LIN {X 0,Y 358.147,Z 231.366,A -85,B 0,C 180,E1 16534.491,E2 16534.491} C_VEL
LIN {X 0,Y 360.808,Z 235.237,A -85,B 0,C 180,E1 16533.457,E2 16533.457} C_VEL
LIN {X 0,Y 363.287,Z 237.581,A -85,B 0,C 180,E1 16532.591,E2 16532.591} C_VEL
LIN {X 0,Y 366.593,Z 241.883,A -85,B 0,C 180,E1 16531.445,E2 16531.445} C_VEL
LIN {X 0,Y 368.213,Z 243.704,A -85,B 0,C 180,E1 16530.917,E2 16530.917} C_VEL
LIN {X 0,Y 371.953,Z 248.281,A -85,B 0,C 180,E1 16529.732,E2 16529.732} C_VEL
LIN {X 0,Y 377.988,Z 256.41,A -85,B 0,C 180,E1 16527.924,E2 16527.924} C_VEL
LIN {X 0,Y 386.57,Z 269.394,A -85,B 0,C 180,E1 16525.541,E2 16525.541} C_VEL
LIN {X 0,Y 395.488,Z 283.924,A -85,B 0,C 180,E1 16523.278,E2 16523.278} C_VEL
LIN {X 0,Y 404.338,Z 299.581,A -85,B 0,C 180,E1 16521.202,E2 16521.202} C_VEL
LIN {X 0,Y 413.977,Z 318.387,A -85,B 0,C 180,E1 16519.091,E2 16519.091} C_VEL
LIN {X 0,Y 416.532,Z 324.265,A -85,B 0,C 180,E1 16518.54,E2 16518.54} C_VEL
LIN {X 0,Y 406.024,Z 519.661,A -85,B 0,C 180,E1 16515.165,E2 16515.165} C_VEL
LIN {X 0,Y 404.264,Z 537.979,A -85,B 0,C 180,E1 16514.727,E2 16514.727} C_VEL
LIN {X 0,Y 401.335,Z 559.6,A -85,B 0,C 180,E1 16514.028,E2 16514.028} C_VEL
LIN {X 0,Y 397.456,Z 581.194,A -85,B 0,C 180,E1 16513.057,E2 16513.057} C_VEL
LIN {X 0,Y 393.804,Z 598.492,A -85,B 0,C 180,E1 16512.084,E2 16512.084} C_VEL
LIN {X 0,Y 389.995,Z 614.356,A -85,B 0,C 180,E1 16511.015,E2 16511.015} C_VEL
LIN {X 0,Y 385.902,Z 629.8,A -85,B 0,C 180,E1 16509.784,E2 16509.784} C_VEL
LIN {X 0,Y 381.564,Z 644.781,A -85,B 0,C 180,E1 16508.387,E2 16508.387} C_VEL
LIN {X 0,Y 376.69,Z 660.514,A -85,B 0,C 180,E1 16506.667,E2 16506.667} C_VEL
LIN {X 0,Y 370.561,Z 678.911,A -85,B 0,C 180,E1 16504.243,E2 16504.243} C_VEL
LIN {X 0,Y 365.986,Z 691.98,A -85,B 0,C 180,E1 16502.186,E2 16502.186} C_VEL
LIN {X 0,Y 361.741,Z 703.869,A -85,B 0,C 180,E1 16500.015,E2 16500.015} C_VEL
LIN {X 0,Y 357.987,Z 714.365,A -85,B 0,C 180,E1 16497.8,E2 16497.8} C_VEL
LIN {X 0,Y 354.508,Z 724.257,A -85,B 0,C 180,E1 16495.382,E2 16495.382} C_VEL
LIN {X 0,Y 351.404,Z 733.441,A -85,B 0,C 180,E1 16492.763,E2 16492.763} C_VEL
LIN {X 0,Y 348.508,Z 742.76,A -85,B 0,C 180,E1 16489.611,E2 16489.611} C_VEL
LIN {X 0,Y 346.148,Z 751.408,A -85,B 0,C 180,E1 16485.925,E2 16485.925} C_VEL
LIN {X 0,Y 344.933,Z 757.022,A -85,B 0,C 180,E1 16482.896,E2 16482.896} C_VEL
LIN {X 0,Y 344.287,Z 761.191,A -85,B 0,C 180,E1 16480.034,E2 16480.034} C_VEL
LIN {X 0,Y 343.998,Z 764.291,A -85,B 0,C 180,E1 16477.179,E2 16477.179} C_VEL
LIN {X 0,Y 343.938,Z 766.265,A -85,B 0,C 180,E1 16474.501,E2 16474.501} C_VEL
LIN {X 0,Y 343.961,Z 767.366,A -85,B 0,C 180,E1 16471.666,E2 16471.666} C_VEL
LIN {X 0,Y 343.968,Z 767.484,A -85,B 0,C 180,E1 16469.001,E2 16469.001} C_VEL
LIN {X 0,Y 343.943,Z 766.62,A -85,B 0,C 180,E1 16466.167,E2 16466.167} C_VEL
LIN {X 0,Y 343.979,Z 764.736,A -85,B 0,C 180,E1 16463.324,E2 16463.324} C_VEL
LIN {X 0,Y 344.211,Z 761.817,A -85,B 0,C 180,E1 16460.47,E2 16460.47} C_VEL
LIN {X 0,Y 344.79,Z 757.833,A -85,B 0,C 180,E1 16457.61,E2 16457.61} C_VEL
LIN {X 0,Y 345.827,Z 752.744,A -85,B 0,C 180,E1 16454.748,E2 16454.748} C_VEL
LIN {X 0,Y 347.309,Z 746.894,A -85,B 0,C 180,E1 16452.061,E2 16452.061} C_VEL
LIN {X 0,Y 349.33,Z 739.94,A -85,B 0,C 180,E1 16449.387,E2 16449.387} C_VEL
LIN {X 0,Y 351.939,Z 731.816,A -85,B 0,C 180,E1 16446.743,E2 16446.743} C_VEL
LIN {X 0,Y 355.383,Z 721.781,A -85,B 0,C 180,E1 16443.969,E2 16443.969} C_VEL
LIN {X 0,Y 360.353,Z 707.827,A -85,B 0,C 180,E1 16440.772,E2 16440.772} C_VEL
LIN {X 0,Y 364.719,Z 695.539,A -85,B 0,C 180,E1 16438.429,E2 16438.429} C_VEL
LIN {X 0,Y 369.153,Z 682.912,A -85,B 0,C 180,E1 16436.358,E2 16436.358} C_VEL
LIN {X 0,Y 373.619,Z 669.807,A -85,B 0,C 180,E1 16434.503,E2 16434.503} C_VEL
LIN {X 0,Y 378.077,Z 656.103,A -85,B 0,C 180,E1 16432.827,E2 16432.827} C_VEL
LIN {X 0,Y 382.633,Z 641.227,A -85,B 0,C 180,E1 16431.261,E2 16431.261} C_VEL
LIN {X 0,Y 387.993,Z 622.392,A -85,B 0,C 180,E1 16429.587,E2 16429.587} C_VEL
LIN {X 0,Y 392.847,Z 602.741,A -85,B 0,C 180,E1 16428.182,E2 16428.182} C_VEL
LIN {X 0,Y 396.506,Z 585.973,A -85,B 0,C 180,E1 16427.194,E2 16427.194} C_VEL
LIN {X 0,Y 399.64,Z 569.419,A -85,B 0,C 180,E1 16426.389,E2 16426.389} C_VEL
LIN {X 0,Y 402.392,Z 552.185,A -85,B 0,C 180,E1 16425.716,E2 16425.716} C_VEL
LIN {X 0,Y 404.611,Z 534.898,A -85,B 0,C 180,E1 16425.192,E2 16425.192} C_VEL
LIN {X 0,Y 406.222,Z 516.887,A -85,B 0,C 180,E1 16424.779,E2 16424.779} C_VEL
LIN {X 0,Y 416.476,Z 323.681,A -85,B 0,C 180,E1 16421.437,E2 16421.437} C_VEL
LIN {X 0,Y 407.354,Z 305.319,A -85,B 0,C 180,E1 16419.475,E2 16419.475} C_VEL
LIN {X 0,Y 397.623,Z 287.545,A -85,B 0,C 180,E1 16417.236,E2 16417.236} C_VEL
LIN {X 0,Y 387.925,Z 271.508,A -85,B 0,C 180,E1 16414.815,E2 16414.815} C_VEL
LIN {X 0,Y 380.179,Z 259.661,A -85,B 0,C 180,E1 16412.707,E2 16412.707} C_VEL
LIN {X 0,Y 375.453,Z 252.882,A -85,B 0,C 180,E1 16411.331,E2 16411.331} C_VEL
LIN {X 0,Y 371.265,Z 247.622,A -85,B 0,C 180,E1 16410.062,E2 16410.062} C_VEL
LIN {X 0,Y 367.142,Z 242.37,A -85,B 0,C 180,E1 16408.731,E2 16408.731} C_VEL
LIN {X 0,Y 363.776,Z 238.413,A -85,B 0,C 180,E1 16407.591,E2 16407.591} C_VEL
LIN {X 0,Y 362.574,Z 236.728,A -85,B 0,C 180,E1 16407.156,E2 16407.156} C_VEL
LIN {X 0,Y 359.338,Z 233.431,A -85,B 0,C 180,E1 16405.993,E2 16405.993} C_VEL
LIN {X 0,Y 357.667,Z 230.823,A -85,B 0,C 180,E1 16405.323,E2 16405.323} C_VEL
LIN {X 0,Y 354.403,Z 228.071,A -85,B 0,C 180,E1 16404.06,E2 16404.06} C_VEL
LIN {X 0,Y 352.382,Z 224.558,A -85,B 0,C 180,E1 16403.141,E2 16403.141} C_VEL
LIN {X 0,Y 348.995,Z 222.277,A -85,B 0,C 180,E1 16401.691,E2 16401.691} C_VEL
LIN {X 0,Y 347.281,Z 219.092,A -85,B 0,C 180,E1 16400.741,E2 16400.741} C_VEL
LIN {X 0,Y 347.017,Z 217.978,A -85,B 0,C 180,E1 16400.053,E2 16400.053} C_VEL
LIN {X 0,Y 347.005,Z 217.928,A -85,B 0,C 180,E1 16395.786,E2 16395.786} C_VEL
LIN {X 0,Y 347.009,Z 217.916,A -85,B 0,C 180,E1 16391.604,E2 16391.604} C_VEL
LIN {X 0,Y 347.012,Z 217.907,A -85,B 0,C 180,E1 16387.45,E2 16387.45} C_VEL
LIN {X 0,Y 347.022,Z 217.907,A -85,B 0,C 180,E1 16383.304,E2 16383.304} C_VEL
LIN {X 0,Y 347.037,Z 217.916,A -85,B 0,C 180,E1 16379.175,E2 16379.175} C_VEL
LIN {X 0,Y 347.034,Z 217.935,A -85,B 0,C 180,E1 16374.876,E2 16374.876} C_VEL
LIN {X 0,Y 347.025,Z 217.934,A -85,B 0,C 180,E1 16370.715,E2 16370.715} C_VEL
LIN {X 0,Y 347.009,Z 217.92,A -85,B 0,C 180,E1 16366.503,E2 16366.503} C_VEL
LIN {X 0,Y 347.007,Z 217.914,A -85,B 0,C 180,E1 16362.389,E2 16362.389} C_VEL
LIN {X 0,Y 347.069,Z 218.147,A -85,B 0,C 180,E1 16359.42,E2 16359.42} C_VEL
LIN {X 0,Y 347.416,Z 219.583,A -85,B 0,C 180,E1 16358.826,E2 16358.826} C_VEL
LIN {X 0,Y 349.081,Z 222.37,A -85,B 0,C 180,E1 16357.961,E2 16357.961} C_VEL
LIN {X 0,Y 352.726,Z 225.069,A -85,B 0,C 180,E1 16356.396,E2 16356.396} C_VEL
LIN {X 0,Y 354.957,Z 228.696,A -85,B 0,C 180,E1 16355.405,E2 16355.405} C_VEL
LIN {X 0,Y 358.15,Z 231.397,A -85,B 0,C 180,E1 16354.181,E2 16354.181} C_VEL
LIN {X 0,Y 360.815,Z 235.248,A -85,B 0,C 180,E1 16353.147,E2 16353.147} C_VEL
LIN {X 0,Y 363.195,Z 237.45,A -85,B 0,C 180,E1 16352.317,E2 16352.317} C_VEL
LIN {X 0,Y 366.384,Z 241.7,A -85,B 0,C 180,E1 16351.205,E2 16351.205} C_VEL
LIN {X 0,Y 368.115,Z 243.592,A -85,B 0,C 180,E1 16350.641,E2 16350.641} C_VEL
LIN {X 0,Y 371.849,Z 248.196,A -85,B 0,C 180,E1 16349.455,E2 16349.455} C_VEL
LIN {X 0,Y 377.907,Z 256.067,A -85,B 0,C 180,E1 16347.647,E2 16347.647} C_VEL
LIN {X 0,Y 384.404,Z 264.582,A -85,B 0,C 180,E1 16345.861,E2 16345.861} C_VEL
LIN {X 0,Y 393.178,Z 275.967,A -85,B 0,C 180,E1 16343.662,E2 16343.662} C_VEL
LIN {X 0,Y 399.805,Z 283.455,A -85,B 0,C 180,E1 16342.167,E2 16342.167} C_VEL
LIN {X 0,Y 407.16,Z 290.873,A -85,B 0,C 180,E1 16340.639,E2 16340.639} C_VEL
LIN {X 0,Y 414.295,Z 297.725,A -85,B 0,C 180,E1 16339.152,E2 16339.152} C_VEL
LIN {X 0,Y 423.422,Z 305.91,A -85,B 0,C 180,E1 16337.148,E2 16337.148} C_VEL
LIN {X 0,Y 430.935,Z 312.908,A -85,B 0,C 180,E1 16335.328,E2 16335.328} C_VEL
LIN {X 0,Y 438.316,Z 319.898,A -85,B 0,C 180,E1 16333.401,E2 16333.401} C_VEL
LIN {X 0,Y 446.153,Z 327.52,A -85,B 0,C 180,E1 16331.147,E2 16331.147} C_VEL
LIN {X 0,Y 453.884,Z 334.907,A -85,B 0,C 180,E1 16328.864,E2 16328.864} C_VEL
LIN {X 0,Y 461.376,Z 342.071,A -85,B 0,C 180,E1 16326.548,E2 16326.548} C_VEL
LIN {X 0,Y 465.487,Z 345.947,A -85,B 0,C 180,E1 16325.234,E2 16325.234} C_VEL
LIN {X 0,Y 472.95,Z 352.634,A -85,B 0,C 180,E1 16322.762,E2 16322.762} C_VEL
LIN {X 0,Y 478.981,Z 358.021,A -85,B 0,C 180,E1 16320.676,E2 16320.676} C_VEL
LIN {X 0,Y 486.038,Z 364.567,A -85,B 0,C 180,E1 16318.048,E2 16318.048} C_VEL
LIN {X 0,Y 490.07,Z 367.772,A -85,B 0,C 180,E1 16316.471,E2 16316.471} C_VEL
LIN {X 0,Y 494.812,Z 372.269,A -85,B 0,C 180,E1 16314.469,E2 16314.469} C_VEL
LIN {X 0,Y 499.341,Z 375.695,A -85,B 0,C 180,E1 16312.483,E2 16312.483} C_VEL
LIN {X 0,Y 503.668,Z 379.96,A -85,B 0,C 180,E1 16310.326,E2 16310.326} C_VEL
LIN {X 0,Y 508.131,Z 382.903,A -85,B 0,C 180,E1 16307.993,E2 16307.993} C_VEL
LIN {X 0,Y 511.92,Z 386.922,A -85,B 0,C 180,E1 16305.635,E2 16305.635} C_VEL
LIN {X 0,Y 515.405,Z 389.563,A -85,B 0,C 180,E1 16303.232,E2 16303.232} C_VEL
LIN {X 0,Y 518.275,Z 391.031,A -85,B 0,C 180,E1 16300.887,E2 16300.887} C_VEL
LIN {X 0,Y 519.23,Z 391.924,A -85,B 0,C 180,E1 16299.979,E2 16299.979} C_VEL
LIN {X 0,Y 521.049,Z 394.222,A -85,B 0,C 180,E1 16297.83,E2 16297.83} C_VEL
LIN {X 0,Y 522.507,Z 395.771,A -85,B 0,C 180,E1 16295.6,E2 16295.6} C_VEL
LIN {X 0,Y 523.67,Z 396.741,A -85,B 0,C 180,E1 16292.955,E2 16292.955} C_VEL
LIN {X 0,Y 524.089,Z 397.007,A -85,B 0,C 180,E1 16290.437,E2 16290.437} C_VEL
LIN {X 0,Y 523.877,Z 396.833,A -85,B 0,C 180,E1 16287.813,E2 16287.813} C_VEL
LIN {X 0,Y 522.974,Z 396.155,A -85,B 0,C 180,E1 16285.285,E2 16285.285} C_VEL
LIN {X 0,Y 521.462,Z 394.714,A -85,B 0,C 180,E1 16282.731,E2 16282.731} C_VEL
LIN {X 0,Y 519.543,Z 392.399,A -85,B 0,C 180,E1 16280.363,E2 16280.363} C_VEL
LIN {X 0,Y 518.399,Z 391.076,A -85,B 0,C 180,E1 16279.218,E2 16279.218} C_VEL
LIN {X 0,Y 515.546,Z 389.656,A -85,B 0,C 180,E1 16276.886,E2 16276.886} C_VEL
LIN {X 0,Y 512.113,Z 387.093,A -85,B 0,C 180,E1 16274.487,E2 16274.487} C_VEL
LIN {X 0,Y 508.669,Z 383.406,A -85,B 0,C 180,E1 16272.323,E2 16272.323} C_VEL
LIN {X 0,Y 503.8,Z 380.064,A -85,B 0,C 180,E1 16269.74,E2 16269.74} C_VEL
LIN {X 0,Y 499.555,Z 375.947,A -85,B 0,C 180,E1 16267.627,E2 16267.627} C_VEL
LIN {X 0,Y 497.104,Z 373.951,A -85,B 0,C 180,E1 16266.523,E2 16266.523} C_VEL
LIN {X 0,Y 492.041,Z 369.824,A -85,B 0,C 180,E1 16264.356,E2 16264.356} C_VEL
LIN {X 0,Y 488.524,Z 366.404,A -85,B 0,C 180,E1 16262.916,E2 16262.916} C_VEL
LIN {X 0,Y 483.274,Z 362.137,A -85,B 0,C 180,E1 16260.912,E2 16260.912} C_VEL
LIN {X 0,Y 478.982,Z 358.023,A -85,B 0,C 180,E1 16259.324,E2 16259.324} C_VEL
LIN {X 0,Y 472.863,Z 352.545,A -85,B 0,C 180,E1 16257.208,E2 16257.208} C_VEL
LIN {X 0,Y 465.164,Z 345.628,A -85,B 0,C 180,E1 16254.662,E2 16254.662} C_VEL
LIN {X 0,Y 461.24,Z 341.963,A -85,B 0,C 180,E1 16253.411,E2 16253.411} C_VEL
LIN {X 0,Y 455.209,Z 336.085,A -85,B 0,C 180,E1 16251.543,E2 16251.543} C_VEL
LIN {X 0,Y 448.292,Z 329.576,A -85,B 0,C 180,E1 16249.467,E2 16249.467} C_VEL
LIN {X 0,Y 440.473,Z 321.942,A -85,B 0,C 180,E1 16247.205,E2 16247.205} C_VEL
LIN {X 0,Y 432.998,Z 314.88,A -85,B 0,C 180,E1 16245.195,E2 16245.195} C_VEL
LIN {X 0,Y 425.304,Z 307.716,A -85,B 0,C 180,E1 16243.307,E2 16243.307} C_VEL
LIN {X 0,Y 416.661,Z 299.751,A -85,B 0,C 180,E1 16241.341,E2 16241.341} C_VEL
LIN {X 0,Y 408.568,Z 292.335,A -85,B 0,C 180,E1 16239.653,E2 16239.653} C_VEL
LIN {X 0,Y 395.556,Z 278.971,A -85,B 0,C 180,E1 16236.895,E2 16236.895} C_VEL
LIN {X 0,Y 384.163,Z 264.207,A -85,B 0,C 180,E1 16234.073,E2 16234.073} C_VEL
LIN {X 0,Y 375.705,Z 253.133,A -85,B 0,C 180,E1 16231.71,E2 16231.71} C_VEL
LIN {X 0,Y 371.276,Z 247.65,A -85,B 0,C 180,E1 16230.373,E2 16230.373} C_VEL
LIN {X 0,Y 367.041,Z 242.298,A -85,B 0,C 180,E1 16229.006,E2 16229.006} C_VEL
LIN {X 0,Y 363.683,Z 238.292,A -85,B 0,C 180,E1 16227.865,E2 16227.865} C_VEL
LIN {X 0,Y 362.476,Z 236.655,A -85,B 0,C 180,E1 16227.43,E2 16227.43} C_VEL
LIN {X 0,Y 359.248,Z 233.319,A -85,B 0,C 180,E1 16226.266,E2 16226.266} C_VEL
LIN {X 0,Y 357.78,Z 230.839,A -85,B 0,C 180,E1 16225.67,E2 16225.67} C_VEL
LIN {X 0,Y 354.592,Z 228.271,A -85,B 0,C 180,E1 16224.444,E2 16224.444} C_VEL
LIN {X 0,Y 352.29,Z 224.536,A -85,B 0,C 180,E1 16223.413,E2 16223.413} C_VEL
LIN {X 0,Y 348.916,Z 222.185,A -85,B 0,C 180,E1 16221.961,E2 16221.961} C_VEL
LIN {X 0,Y 347.308,Z 219.24,A -85,B 0,C 180,E1 16221.092,E2 16221.092} C_VEL
LIN {X 0,Y 347.038,Z 218.008,A -85,B 0,C 180,E1 16220.403,E2 16220.403} C_VEL
LIN {X 0,Y 347.011,Z 217.912,A -85,B 0,C 180,E1 16216.23,E2 16216.23} C_VEL
LIN {X 0,Y 347.007,Z 217.907,A -85,B 0,C 180,E1 16212.143,E2 16212.143} C_VEL
LIN {X 0,Y 347.004,Z 217.91,A -85,B 0,C 180,E1 16207.95,E2 16207.95} C_VEL
LIN {X 0,Y 347.037,Z 217.938,A -85,B 0,C 180,E1 16204.997,E2 16204.997} C_VEL
LIN {X 0,Y 346.181,Z 218.071,A -85,B 0,C 180,E1 16203.814,E2 16203.814} C_VEL
LIN {X 0,Y 342.295,Z 218.566,A -85,B 0,C 180,E1 16201.771,E2 16201.771} C_VEL
LIN {X 0,Y 339.403,Z 218.9,A -85,B 0,C 180,E1 16199.944,E2 16199.944} C_VEL
LIN {X 0,Y 339.099,Z 218.919,A -85,B 0,C 180,E1 16199.189,E2 16199.189} C_VEL
LIN {X 0,Y 339.096,Z 218.918,A -85,B 0,C 180,E1 16194.925,E2 16194.925} C_VEL
LIN {X 0,Y 339.091,Z 218.899,A -85,B 0,C 180,E1 16190.838,E2 16190.838} C_VEL
LIN {X 0,Y 339.071,Z 218.899,A -85,B 0,C 180,E1 16186.528,E2 16186.528} C_VEL
LIN {X 0,Y 339.135,Z 219.241,A -85,B 0,C 180,E1 16183.558,E2 16183.558} C_VEL
LIN {X 0,Y 339.495,Z 220.608,A -85,B 0,C 180,E1 16182.871,E2 16182.871} C_VEL
LIN {X 0,Y 341.139,Z 223.342,A -85,B 0,C 180,E1 16181.811,E2 16181.811} C_VEL
LIN {X 0,Y 345.112,Z 226.275,A -85,B 0,C 180,E1 16179.743,E2 16179.743} C_VEL
LIN {X 0,Y 347.047,Z 229.639,A -85,B 0,C 180,E1 16178.714,E2 16178.714} C_VEL
LIN {X 0,Y 350.515,Z 232.379,A -85,B 0,C 180,E1 16177.172,E2 16177.172} C_VEL
LIN {X 0,Y 352.892,Z 236.07,A -85,B 0,C 180,E1 16176.098,E2 16176.098} C_VEL
LIN {X 0,Y 355.926,Z 238.789,A -85,B 0,C 180,E1 16174.9,E2 16174.9} C_VEL
LIN {X 0,Y 358.959,Z 242.898,A -85,B 0,C 180,E1 16173.711,E2 16173.711} C_VEL
LIN {X 0,Y 360.889,Z 244.817,A -85,B 0,C 180,E1 16173.019,E2 16173.019} C_VEL
LIN {X 0,Y 364.473,Z 249.345,A -85,B 0,C 180,E1 16171.755,E2 16171.755} C_VEL
LIN {X 0,Y 370.627,Z 257.201,A -85,B 0,C 180,E1 16169.747,E2 16169.747} C_VEL
LIN {X 0,Y 374.807,Z 262.798,A -85,B 0,C 180,E1 16168.474,E2 16168.474} C_VEL
LIN {X 0,Y 383.24,Z 275.79,A -85,B 0,C 180,E1 16166.059,E2 16166.059} C_VEL
LIN {X 0,Y 391.955,Z 290.261,A -85,B 0,C 180,E1 16163.78,E2 16163.78} C_VEL
LIN {X 0,Y 400.678,Z 305.953,A -85,B 0,C 180,E1 16161.674,E2 16161.674} C_VEL
LIN {X 0,Y 409.906,Z 324.383,A -85,B 0,C 180,E1 16159.59,E2 16159.59} C_VEL
LIN {X 0,Y 411.081,Z 327.304,A -85,B 0,C 180,E1 16159.323,E2 16159.323} C_VEL
LIN {X 0,Y 400.412,Z 519.486,A -85,B 0,C 180,E1 16155.979,E2 16155.979} C_VEL
LIN {X 0,Y 398.606,Z 537.803,A -85,B 0,C 180,E1 16155.538,E2 16155.538} C_VEL
LIN {X 0,Y 395.601,Z 559.424,A -85,B 0,C 180,E1 16154.836,E2 16154.836} C_VEL
LIN {X 0,Y 391.654,Z 580.821,A -85,B 0,C 180,E1 16153.871,E2 16153.871} C_VEL
LIN {X 0,Y 387.858,Z 598.316,A -85,B 0,C 180,E1 16152.882,E2 16152.882} C_VEL
LIN {X 0,Y 383.939,Z 614.18,A -85,B 0,C 180,E1 16151.806,E2 16151.806} C_VEL
LIN {X 0,Y 379.721,Z 629.623,A -85,B 0,C 180,E1 16150.565,E2 16150.565} C_VEL
LIN {X 0,Y 375.244,Z 644.604,A -85,B 0,C 180,E1 16149.156,E2 16149.156} C_VEL
LIN {X 0,Y 370.205,Z 660.337,A -85,B 0,C 180,E1 16147.418,E2 16147.418} C_VEL
LIN {X 0,Y 363.831,Z 678.801,A -85,B 0,C 180,E1 16144.955,E2 16144.955} C_VEL
LIN {X 0,Y 359.109,Z 691.802,A -85,B 0,C 180,E1 16142.88,E2 16142.88} C_VEL
LIN {X 0,Y 354.693,Z 703.69,A -85,B 0,C 180,E1 16140.675,E2 16140.675} C_VEL
LIN {X 0,Y 350.777,Z 714.186,A -85,B 0,C 180,E1 16138.422,E2 16138.422} C_VEL
LIN {X 0,Y 347.134,Z 724.078,A -85,B 0,C 180,E1 16135.961,E2 16135.961} C_VEL
LIN {X 0,Y 343.877,Z 733.263,A -85,B 0,C 180,E1 16133.29,E2 16133.29} C_VEL
LIN {X 0,Y 340.825,Z 742.581,A -85,B 0,C 180,E1 16130.072,E2 16130.072} C_VEL
LIN {X 0,Y 338.32,Z 751.23,A -85,B 0,C 180,E1 16126.304,E2 16126.304} C_VEL
LIN {X 0,Y 337.022,Z 756.844,A -85,B 0,C 180,E1 16123.204,E2 16123.204} C_VEL
LIN {X 0,Y 336.316,Z 761.063,A -85,B 0,C 180,E1 16120.233,E2 16120.233} C_VEL
LIN {X 0,Y 336.008,Z 764.115,A -85,B 0,C 180,E1 16117.351,E2 16117.351} C_VEL
LIN {X 0,Y 335.938,Z 766.09,A -85,B 0,C 180,E1 16114.609,E2 16114.609} C_VEL
LIN {X 0,Y 335.963,Z 767.191,A -85,B 0,C 180,E1 16111.705,E2 16111.705} C_VEL
LIN {X 0,Y 335.969,Z 767.309,A -85,B 0,C 180,E1 16108.977,E2 16108.977} C_VEL
LIN {X 0,Y 335.944,Z 766.445,A -85,B 0,C 180,E1 16106.075,E2 16106.075} C_VEL
LIN {X 0,Y 335.983,Z 764.56,A -85,B 0,C 180,E1 16103.164,E2 16103.164} C_VEL
LIN {X 0,Y 336.243,Z 761.64,A -85,B 0,C 180,E1 16100.242,E2 16100.242} C_VEL
LIN {X 0,Y 336.865,Z 757.656,A -85,B 0,C 180,E1 16097.313,E2 16097.313} C_VEL
LIN {X 0,Y 337.976,Z 752.566,A -85,B 0,C 180,E1 16094.384,E2 16094.384} C_VEL
LIN {X 0,Y 339.672,Z 746.316,A -85,B 0,C 180,E1 16091.465,E2 16091.465} C_VEL
LIN {X 0,Y 342,Z 738.83,A -85,B 0,C 180,E1 16088.567,E2 16088.567} C_VEL
LIN {X 0,Y 345.639,Z 728.384,A -85,B 0,C 180,E1 16085.203,E2 16085.203} C_VEL
LIN {X 0,Y 350.004,Z 716.291,A -85,B 0,C 180,E1 16082.066,E2 16082.066} C_VEL
LIN {X 0,Y 354.099,Z 705.273,A -85,B 0,C 180,E1 16079.643,E2 16079.643} C_VEL
LIN {X 0,Y 358.446,Z 693.581,A -85,B 0,C 180,E1 16077.432,E2 16077.432} C_VEL
LIN {X 0,Y 363.101,Z 680.798,A -85,B 0,C 180,E1 16075.349,E2 16075.349} C_VEL
LIN {X 0,Y 368.01,Z 666.826,A -85,B 0,C 180,E1 16073.394,E2 16073.394} C_VEL
LIN {X 0,Y 374.172,Z 648.158,A -85,B 0,C 180,E1 16071.203,E2 16071.203} C_VEL
LIN {X 0,Y 379.265,Z 631.234,A -85,B 0,C 180,E1 16069.574,E2 16069.574} C_VEL
LIN {X 0,Y 383.699,Z 615.1,A -85,B 0,C 180,E1 16068.262,E2 16068.262} C_VEL
LIN {X 0,Y 387.611,Z 599.378,A -85,B 0,C 180,E1 16067.185,E2 16067.185} C_VEL
LIN {X 0,Y 391.143,Z 583.308,A -85,B 0,C 180,E1 16066.26,E2 16066.26} C_VEL
LIN {X 0,Y 394.27,Z 566.931,A -85,B 0,C 180,E1 16065.483,E2 16065.483} C_VEL
LIN {X 0,Y 397.038,Z 549.662,A -85,B 0,C 180,E1 16064.826,E2 16064.826} C_VEL
LIN {X 0,Y 399.578,Z 529.4,A -85,B 0,C 180,E1 16064.239,E2 16064.239} C_VEL
LIN {X 0,Y 401.626,Z 499.971,A -85,B 0,C 180,E1 16063.654,E2 16063.654} C_VEL
LIN {X 0,Y 410.98,Z 326.671,A -85,B 0,C 180,E1 16060.644,E2 16060.644} C_VEL
LIN {X 0,Y 401.925,Z 308.398,A -85,B 0,C 180,E1 16058.618,E2 16058.618} C_VEL
LIN {X 0,Y 393.275,Z 292.56,A -85,B 0,C 180,E1 16056.549,E2 16056.549} C_VEL
LIN {X 0,Y 384.33,Z 277.523,A -85,B 0,C 180,E1 16054.237,E2 16054.237} C_VEL
LIN {X 0,Y 376.98,Z 266.097,A -85,B 0,C 180,E1 16052.172,E2 16052.172} C_VEL
LIN {X 0,Y 372.654,Z 259.767,A -85,B 0,C 180,E1 16050.874,E2 16050.874} C_VEL
LIN {X 0,Y 368.42,Z 254.411,A -85,B 0,C 180,E1 16049.556,E2 16049.556} C_VEL
LIN {X 0,Y 364.365,Z 249.243,A -85,B 0,C 180,E1 16048.209,E2 16048.209} C_VEL
LIN {X 0,Y 360.793,Z 244.653,A -85,B 0,C 180,E1 16046.944,E2 16046.944} C_VEL
LIN {X 0,Y 356.739,Z 240.167,A -85,B 0,C 180,E1 16045.439,E2 16045.439} C_VEL
LIN {X 0,Y 355.359,Z 238.154,A -85,B 0,C 180,E1 16044.876,E2 16044.876} C_VEL
LIN {X 0,Y 352.004,Z 234.978,A -85,B 0,C 180,E1 16043.522,E2 16043.522} C_VEL
LIN {X 0,Y 350.169,Z 232.005,A -85,B 0,C 180,E1 16042.674,E2 16042.674} C_VEL
LIN {X 0,Y 346.887,Z 229.448,A -85,B 0,C 180,E1 16041.208,E2 16041.208} C_VEL
LIN {X 0,Y 344.663,Z 225.657,A -85,B 0,C 180,E1 16040.019,E2 16040.019} C_VEL
LIN {X 0,Y 341.139,Z 223.339,A -85,B 0,C 180,E1 16038.189,E2 16038.189} C_VEL
LIN {X 0,Y 339.459,Z 220.497,A -85,B 0,C 180,E1 16037.098,E2 16037.098} C_VEL
LIN {X 0,Y 339.135,Z 219.241,A -85,B 0,C 180,E1 16036.442,E2 16036.442} C_VEL
LIN {X 0,Y 339.098,Z 218.89,A -85,B 0,C 180,E1 16032.777,E2 16032.777} C_VEL
LIN {X 0,Y 339.08,Z 218.894,A -85,B 0,C 180,E1 16028.479,E2 16028.479} C_VEL
LIN {X 0,Y 339.069,Z 218.907,A -85,B 0,C 180,E1 16024.228,E2 16024.228} C_VEL
LIN {X 0,Y 339.067,Z 218.922,A -85,B 0,C 180,E1 16019.831,E2 16019.831} C_VEL
LIN {X 0,Y 339.075,Z 218.926,A -85,B 0,C 180,E1 16015.603,E2 16015.603} C_VEL
LIN {X 0,Y 339.091,Z 218.906,A -85,B 0,C 180,E1 16011.351,E2 16011.351} C_VEL
LIN {X 0,Y 339.099,Z 218.898,A -85,B 0,C 180,E1 16007.05,E2 16007.05} C_VEL
LIN {X 0,Y 339.131,Z 219.155,A -85,B 0,C 180,E1 16003.355,E2 16003.355} C_VEL
LIN {X 0,Y 339.438,Z 220.483,A -85,B 0,C 180,E1 16002.608,E2 16002.608} C_VEL
LIN {X 0,Y 341.072,Z 223.266,A -85,B 0,C 180,E1 16001.542,E2 16001.542} C_VEL
LIN {X 0,Y 344.098,Z 225.398,A -85,B 0,C 180,E1 15999.947,E2 15999.947} C_VEL
LIN {X 0,Y 345.044,Z 226.147,A -85,B 0,C 180,E1 15999.473,E2 15999.473} C_VEL
LIN {X 0,Y 346.971,Z 229.551,A -85,B 0,C 180,E1 15998.443,E2 15998.443} C_VEL
LIN {X 0,Y 350.604,Z 232.521,A -85,B 0,C 180,E1 15996.824,E2 15996.824} C_VEL
LIN {X 0,Y 353.175,Z 236.354,A -85,B 0,C 180,E1 15995.674,E2 15995.674} C_VEL
LIN {X 0,Y 355.931,Z 238.825,A -85,B 0,C 180,E1 15994.589,E2 15994.589} C_VEL
LIN {X 0,Y 358.868,Z 242.812,A -85,B 0,C 180,E1 15993.436,E2 15993.436} C_VEL
LIN {X 0,Y 360.896,Z 244.86,A -85,B 0,C 180,E1 15992.708,E2 15992.708} C_VEL
LIN {X 0,Y 364.375,Z 249.269,A -85,B 0,C 180,E1 15991.479,E2 15991.479} C_VEL
LIN {X 0,Y 370.642,Z 257.217,A -85,B 0,C 180,E1 15989.435,E2 15989.435} C_VEL
LIN {X 0,Y 377.776,Z 266.384,A -85,B 0,C 180,E1 15987.32,E2 15987.32} C_VEL
LIN {X 0,Y 390.012,Z 282.705,A -85,B 0,C 180,E1 15984.094,E2 15984.094} C_VEL
LIN {X 0,Y 400.852,Z 294.887,A -85,B 0,C 180,E1 15981.648,E2 15981.648} C_VEL
LIN {X 0,Y 411.801,Z 305.121,A -85,B 0,C 180,E1 15979.403,E2 15979.403} C_VEL
LIN {X 0,Y 420.346,Z 312.786,A -85,B 0,C 180,E1 15977.548,E2 15977.548} C_VEL
LIN {X 0,Y 428.931,Z 320.521,A -85,B 0,C 180,E1 15975.533,E2 15975.533} C_VEL
LIN {X 0,Y 436.134,Z 327.314,A -85,B 0,C 180,E1 15973.67,E2 15973.67} C_VEL
LIN {X 0,Y 443.833,Z 334.746,A -85,B 0,C 180,E1 15971.49,E2 15971.49} C_VEL
LIN {X 0,Y 451.846,Z 342.342,A -85,B 0,C 180,E1 15969.138,E2 15969.138} C_VEL
LIN {X 0,Y 459.256,Z 349.418,A -85,B 0,C 180,E1 15966.858,E2 15966.858} C_VEL
LIN {X 0,Y 463.223,Z 353.072,A -85,B 0,C 180,E1 15965.607,E2 15965.607} C_VEL
LIN {X 0,Y 469.315,Z 358.377,A -85,B 0,C 180,E1 15963.632,E2 15963.632} C_VEL
LIN {X 0,Y 476.158,Z 364.766,A -85,B 0,C 180,E1 15961.277,E2 15961.277} C_VEL
LIN {X 0,Y 479.829,Z 367.961,A -85,B 0,C 180,E1 15959.968,E2 15959.968} C_VEL
LIN {X 0,Y 485.446,Z 373,A -85,B 0,C 180,E1 15957.872,E2 15957.872} C_VEL
LIN {X 0,Y 488.703,Z 375.613,A -85,B 0,C 180,E1 15956.606,E2 15956.606} C_VEL
LIN {X 0,Y 493.806,Z 380.339,A -85,B 0,C 180,E1 15954.458,E2 15954.458} C_VEL
LIN {X 0,Y 498.032,Z 383.54,A -85,B 0,C 180,E1 15952.608,E2 15952.608} C_VEL
LIN {X 0,Y 502.49,Z 387.851,A -85,B 0,C 180,E1 15950.408,E2 15950.408} C_VEL
LIN {X 0,Y 506.98,Z 390.784,A -85,B 0,C 180,E1 15948.079,E2 15948.079} C_VEL
LIN {X 0,Y 510.675,Z 394.71,A -85,B 0,C 180,E1 15945.791,E2 15945.791} C_VEL
LIN {X 0,Y 514.032,Z 397.299,A -85,B 0,C 180,E1 15943.497,E2 15943.497} C_VEL
LIN {X 0,Y 517.12,Z 398.912,A -85,B 0,C 180,E1 15941.034,E2 15941.034} C_VEL
LIN {X 0,Y 518.123,Z 399.754,A -85,B 0,C 180,E1 15940.113,E2 15940.113} C_VEL
LIN {X 0,Y 519.976,Z 402.085,A -85,B 0,C 180,E1 15937.957,E2 15937.957} C_VEL
LIN {X 0,Y 521.451,Z 403.659,A -85,B 0,C 180,E1 15935.722,E2 15935.722} C_VEL
LIN {X 0,Y 522.676,Z 404.668,A -85,B 0,C 180,E1 15933.03,E2 15933.03} C_VEL
LIN {X 0,Y 523.103,Z 404.947,A -85,B 0,C 180,E1 15930.548,E2 15930.548} C_VEL
LIN {X 0,Y 522.899,Z 404.775,A -85,B 0,C 180,E1 15927.809,E2 15927.809} C_VEL
LIN {X 0,Y 522.043,Z 404.137,A -85,B 0,C 180,E1 15925.387,E2 15925.387} C_VEL
LIN {X 0,Y 520.471,Z 402.67,A -85,B 0,C 180,E1 15922.717,E2 15922.717} C_VEL
LIN {X 0,Y 518.536,Z 400.38,A -85,B 0,C 180,E1 15920.344,E2 15920.344} C_VEL
LIN {X 0,Y 517.388,Z 399.01,A -85,B 0,C 180,E1 15919.197,E2 15919.197} C_VEL
LIN {X 0,Y 514.486,Z 397.567,A -85,B 0,C 180,E1 15916.826,E2 15916.826} C_VEL
LIN {X 0,Y 511.058,Z 395.05,A -85,B 0,C 180,E1 15914.454,E2 15914.454} C_VEL
LIN {X 0,Y 507.587,Z 391.429,A -85,B 0,C 180,E1 15912.284,E2 15912.284} C_VEL
LIN {X 0,Y 502.56,Z 387.906,A -85,B 0,C 180,E1 15909.627,E2 15909.627} C_VEL
LIN {X 0,Y 498.11,Z 383.621,A -85,B 0,C 180,E1 15907.427,E2 15907.427} C_VEL
LIN {X 0,Y 495.022,Z 381.224,A -85,B 0,C 180,E1 15906.05,E2 15906.05} C_VEL
LIN {X 0,Y 489.902,Z 376.889,A -85,B 0,C 180,E1 15903.902,E2 15903.902} C_VEL
LIN {X 0,Y 486.672,Z 373.888,A -85,B 0,C 180,E1 15902.603,E2 15902.603} C_VEL
LIN {X 0,Y 481.097,Z 369.232,A -85,B 0,C 180,E1 15900.495,E2 15900.495} C_VEL
LIN {X 0,Y 477.224,Z 365.597,A -85,B 0,C 180,E1 15899.089,E2 15899.089} C_VEL
LIN {X 0,Y 471.197,Z 360.208,A -85,B 0,C 180,E1 15897.006,E2 15897.006} C_VEL
LIN {X 0,Y 463.479,Z 353.332,A -85,B 0,C 180,E1 15894.476,E2 15894.476} C_VEL
LIN {X 0,Y 459.476,Z 349.597,A -85,B 0,C 180,E1 15893.209,E2 15893.209} C_VEL
LIN {X 0,Y 453.383,Z 343.732,A -85,B 0,C 180,E1 15891.326,E2 15891.326} C_VEL
LIN {X 0,Y 446.057,Z 336.852,A -85,B 0,C 180,E1 15889.151,E2 15889.151} C_VEL
LIN {X 0,Y 438.328,Z 329.378,A -85,B 0,C 180,E1 15886.932,E2 15886.932} C_VEL
LIN {X 0,Y 430.853,Z 322.447,A -85,B 0,C 180,E1 15884.964,E2 15884.964} C_VEL
LIN {X 0,Y 421.95,Z 314.119,A -85,B 0,C 180,E1 15882.805,E2 15882.805} C_VEL
LIN {X 0,Y 414.154,Z 307.212,A -85,B 0,C 180,E1 15881.094,E2 15881.094} C_VEL
LIN {X 0,Y 405.719,Z 299.518,A -85,B 0,C 180,E1 15879.345,E2 15879.345} C_VEL
LIN {X 0,Y 392.1,Z 285.378,A -85,B 0,C 180,E1 15876.408,E2 15876.408} C_VEL
LIN {X 0,Y 380.878,Z 270.599,A -85,B 0,C 180,E1 15873.546,E2 15873.546} C_VEL
LIN {X 0,Y 372.442,Z 259.51,A -85,B 0,C 180,E1 15871.118,E2 15871.118} C_VEL
LIN {X 0,Y 368.432,Z 254.445,A -85,B 0,C 180,E1 15869.868,E2 15869.868} C_VEL
LIN {X 0,Y 364.268,Z 249.165,A -85,B 0,C 180,E1 15868.485,E2 15868.485} C_VEL
LIN {X 0,Y 360.704,Z 244.531,A -85,B 0,C 180,E1 15867.219,E2 15867.219} C_VEL
LIN {X 0,Y 356.745,Z 240.197,A -85,B 0,C 180,E1 15865.75,E2 15865.75} C_VEL
LIN {X 0,Y 355.469,Z 238.2,A -85,B 0,C 180,E1 15865.224,E2 15865.224} C_VEL
LIN {X 0,Y 352.189,Z 235.184,A -85,B 0,C 180,E1 15863.909,E2 15863.909} C_VEL
LIN {X 0,Y 350.265,Z 232.073,A -85,B 0,C 180,E1 15863.022,E2 15863.022} C_VEL
LIN {X 0,Y 346.812,Z 229.356,A -85,B 0,C 180,E1 15861.479,E2 15861.479} C_VEL
LIN {X 0,Y 344.588,Z 225.599,A -85,B 0,C 180,E1 15860.289,E2 15860.289} C_VEL
LIN {X 0,Y 341.354,Z 223.556,A -85,B 0,C 180,E1 15858.619,E2 15858.619} C_VEL
LIN {X 0,Y 339.542,Z 220.78,A -85,B 0,C 180,E1 15857.48,E2 15857.48} C_VEL
LIN {X 0,Y 339.155,Z 219.267,A -85,B 0,C 180,E1 15856.793,E2 15856.793} C_VEL
LIN {X 0,Y 339.077,Z 218.923,A -85,B 0,C 180,E1 15854.342,E2 15854.342} C_VEL
LIN {X 0,Y 339.069,Z 218.926,A -85,B 0,C 180,E1 15850.02,E2 15850.02} C_VEL
LIN {X 0,Y 339.065,Z 218.911,A -85,B 0,C 180,E1 15845.754,E2 15845.754} C_VEL
LIN {X 0,Y 339.074,Z 218.897,A -85,B 0,C 180,E1 15841.521,E2 15841.521} C_VEL
LIN {X 0,Y 339.099,Z 218.919,A -85,B 0,C 180,E1 15839.189,E2 15839.189} C_VEL
LIN {X 0,Y 338.281,Z 219,A -85,B 0,C 180,E1 15837.979,E2 15837.979} C_VEL
LIN {X 0,Y 334.574,Z 219.466,A -85,B 0,C 180,E1 15835.98,E2 15835.98} C_VEL
LIN {X 0,Y 331.467,Z 219.863,A -85,B 0,C 180,E1 15834.017,E2 15834.017} C_VEL
LIN {X 0,Y 331.161,Z 219.885,A -85,B 0,C 180,E1 15833.244,E2 15833.244} C_VEL
LIN {X 0,Y 331.179,Z 220.067,A -85,B 0,C 180,E1 15829.211,E2 15829.211} C_VEL
LIN {X 0,Y 331.471,Z 221.413,A -85,B 0,C 180,E1 15828.031,E2 15828.031} C_VEL
LIN {X 0,Y 333.583,Z 224.73,A -85,B 0,C 180,E1 15826.125,E2 15826.125} C_VEL
LIN {X 0,Y 337.44,Z 227.336,A -85,B 0,C 180,E1 15823.517,E2 15823.517} C_VEL
LIN {X 0,Y 339.207,Z 230.574,A -85,B 0,C 180,E1 15822.325,E2 15822.325} C_VEL
LIN {X 0,Y 342.761,Z 233.257,A -85,B 0,C 180,E1 15820.398,E2 15820.398} C_VEL
LIN {X 0,Y 345.759,Z 237.709,A -85,B 0,C 180,E1 15818.808,E2 15818.808} C_VEL
LIN {X 0,Y 348.577,Z 240.082,A -85,B 0,C 180,E1 15817.528,E2 15817.528} C_VEL
LIN {X 0,Y 351.392,Z 244.003,A -85,B 0,C 180,E1 15816.256,E2 15816.256} C_VEL
LIN {X 0,Y 353.818,Z 246.306,A -85,B 0,C 180,E1 15815.276,E2 15815.276} C_VEL
LIN {X 0,Y 357.219,Z 250.639,A -85,B 0,C 180,E1 15813.93,E2 15813.93} C_VEL
LIN {X 0,Y 358.898,Z 252.633,A -85,B 0,C 180,E1 15813.305,E2 15813.305} C_VEL
LIN {X 0,Y 363.49,Z 258.436,A -85,B 0,C 180,E1 15811.672,E2 15811.672} C_VEL
LIN {X 0,Y 368.43,Z 264.838,A -85,B 0,C 180,E1 15810.042,E2 15810.042} C_VEL
LIN {X 0,Y 371.882,Z 269.556,A -85,B 0,C 180,E1 15808.965,E2 15808.965} C_VEL
LIN {X 0,Y 379.942,Z 282.185,A -85,B 0,C 180,E1 15806.586,E2 15806.586} C_VEL
LIN {X 0,Y 388.328,Z 296.367,A -85,B 0,C 180,E1 15804.323,E2 15804.323} C_VEL
LIN {X 0,Y 397.045,Z 312.321,A -85,B 0,C 180,E1 15802.155,E2 15802.155} C_VEL
LIN {X 0,Y 405.723,Z 330.052,A -85,B 0,C 180,E1 15800.132,E2 15800.132} C_VEL
LIN {X 0,Y 394.88,Z 519.316,A -85,B 0,C 180,E1 15796.816,E2 15796.816} C_VEL
LIN {X 0,Y 393.032,Z 537.628,A -85,B 0,C 180,E1 15796.372,E2 15796.372} C_VEL
LIN {X 0,Y 389.947,Z 559.249,A -85,B 0,C 180,E1 15795.668,E2 15795.668} C_VEL
LIN {X 0,Y 385.893,Z 580.645,A -85,B 0,C 180,E1 15794.699,E2 15794.699} C_VEL
LIN {X 0,Y 381.991,Z 598.14,A -85,B 0,C 180,E1 15793.705,E2 15793.705} C_VEL
LIN {X 0,Y 377.959,Z 614.003,A -85,B 0,C 180,E1 15792.622,E2 15792.622} C_VEL
LIN {X 0,Y 373.613,Z 629.446,A -85,B 0,C 180,E1 15791.372,E2 15791.372} C_VEL
LIN {X 0,Y 368.996,Z 644.427,A -85,B 0,C 180,E1 15789.95,E2 15789.95} C_VEL
LIN {X 0,Y 363.68,Z 660.483,A -85,B 0,C 180,E1 15788.157,E2 15788.157} C_VEL
LIN {X 0,Y 357.315,Z 678.286,A -85,B 0,C 180,E1 15785.755,E2 15785.755} C_VEL
LIN {X 0,Y 352.287,Z 691.623,A -85,B 0,C 180,E1 15783.6,E2 15783.6} C_VEL
LIN {X 0,Y 347.694,Z 703.512,A -85,B 0,C 180,E1 15781.362,E2 15781.362} C_VEL
LIN {X 0,Y 343.61,Z 714.008,A -85,B 0,C 180,E1 15779.071,E2 15779.071} C_VEL
LIN {X 0,Y 339.757,Z 724.011,A -85,B 0,C 180,E1 15776.535,E2 15776.535} C_VEL
LIN {X 0,Y 336.38,Z 733.084,A -85,B 0,C 180,E1 15773.841,E2 15773.841} C_VEL
LIN {X 0,Y 333.152,Z 742.434,A -85,B 0,C 180,E1 15770.542,E2 15770.542} C_VEL
LIN {X 0,Y 330.507,Z 751.052,A -85,B 0,C 180,E1 15766.7,E2 15766.7} C_VEL
LIN {X 0,Y 329.119,Z 756.667,A -85,B 0,C 180,E1 15763.527,E2 15763.527} C_VEL
LIN {X 0,Y 328.36,Z 760.837,A -85,B 0,C 180,E1 15760.526,E2 15760.526} C_VEL
LIN {X 0,Y 328.02,Z 763.939,A -85,B 0,C 180,E1 15757.531,E2 15757.531} C_VEL
LIN {X 0,Y 327.938,Z 765.914,A -85,B 0,C 180,E1 15754.721,E2 15754.721} C_VEL
LIN {X 0,Y 327.963,Z 766.987,A -85,B 0,C 180,E1 15751.922,E2 15751.922} C_VEL
LIN {X 0,Y 327.97,Z 767.135,A -85,B 0,C 180,E1 15748.952,E2 15748.952} C_VEL
LIN {X 0,Y 327.945,Z 766.269,A -85,B 0,C 180,E1 15745.979,E2 15745.979} C_VEL
LIN {X 0,Y 327.989,Z 764.384,A -85,B 0,C 180,E1 15742.997,E2 15742.997} C_VEL
LIN {X 0,Y 328.277,Z 761.464,A -85,B 0,C 180,E1 15740.003,E2 15740.003} C_VEL
LIN {X 0,Y 328.948,Z 757.478,A -85,B 0,C 180,E1 15737.003,E2 15737.003} C_VEL
LIN {X 0,Y 330.139,Z 752.388,A -85,B 0,C 180,E1 15734.004,E2 15734.004} C_VEL
LIN {X 0,Y 331.942,Z 746.137,A -85,B 0,C 180,E1 15731.018,E2 15731.018} C_VEL
LIN {X 0,Y 334.404,Z 738.651,A -85,B 0,C 180,E1 15728.056,E2 15728.056} C_VEL
LIN {X 0,Y 338.232,Z 728.205,A -85,B 0,C 180,E1 15724.622,E2 15724.622} C_VEL
LIN {X 0,Y 342.888,Z 715.884,A -85,B 0,C 180,E1 15721.372,E2 15721.372} C_VEL
LIN {X 0,Y 347.076,Z 705.095,A -85,B 0,C 180,E1 15718.962,E2 15718.962} C_VEL
LIN {X 0,Y 351.599,Z 693.403,A -85,B 0,C 180,E1 15716.716,E2 15716.716} C_VEL
LIN {X 0,Y 356.43,Z 680.62,A -85,B 0,C 180,E1 15714.605,E2 15714.605} C_VEL
LIN {X 0,Y 361.434,Z 666.872,A -85,B 0,C 180,E1 15712.656,E2 15712.656} C_VEL
LIN {X 0,Y 367.667,Z 648.692,A -85,B 0,C 180,E1 15710.484,E2 15710.484} C_VEL
LIN {X 0,Y 373.142,Z 631.057,A -85,B 0,C 180,E1 15708.769,E2 15708.769} C_VEL
LIN {X 0,Y 377.712,Z 614.923,A -85,B 0,C 180,E1 15707.447,E2 15707.447} C_VEL
LIN {X 0,Y 381.737,Z 599.202,A -85,B 0,C 180,E1 15706.362,E2 15706.362} C_VEL
LIN {X 0,Y 385.367,Z 583.132,A -85,B 0,C 180,E1 15705.432,E2 15705.432} C_VEL
LIN {X 0,Y 388.58,Z 566.756,A -85,B 0,C 180,E1 15704.652,E2 15704.652} C_VEL
LIN {X 0,Y 391.434,Z 549.422,A -85,B 0,C 180,E1 15703.991,E2 15703.991} C_VEL
LIN {X 0,Y 394.061,Z 528.93,A -85,B 0,C 180,E1 15703.396,E2 15703.396} C_VEL
LIN {X 0,Y 396.16,Z 499.287,A -85,B 0,C 180,E1 15702.806,E2 15702.806} C_VEL
LIN {X 0,Y 405.601,Z 329.786,A -85,B 0,C 180,E1 15699.84,E2 15699.84} C_VEL
LIN {X 0,Y 396.589,Z 311.477,A -85,B 0,C 180,E1 15697.737,E2 15697.737} C_VEL
LIN {X 0,Y 387.405,Z 294.658,A -85,B 0,C 180,E1 15695.434,E2 15695.434} C_VEL
LIN {X 0,Y 377.48,Z 278.167,A -85,B 0,C 180,E1 15692.709,E2 15692.709} C_VEL
LIN {X 0,Y 369.993,Z 266.78,A -85,B 0,C 180,E1 15690.445,E2 15690.445} C_VEL
LIN {X 0,Y 365.28,Z 260.808,A -85,B 0,C 180,E1 15688.936,E2 15688.936} C_VEL
LIN {X 0,Y 361.727,Z 256.185,A -85,B 0,C 180,E1 15687.716,E2 15687.716} C_VEL
LIN {X 0,Y 357.42,Z 250.822,A -85,B 0,C 180,E1 15686.143,E2 15686.143} C_VEL
LIN {X 0,Y 353.995,Z 246.606,A -85,B 0,C 180,E1 15684.8,E2 15684.8} C_VEL
LIN {X 0,Y 352.885,Z 245.307,A -85,B 0,C 180,E1 15684.348,E2 15684.348} C_VEL
LIN {X 0,Y 349.47,Z 241.621,A -85,B 0,C 180,E1 15682.9,E2 15682.9} C_VEL
LIN {X 0,Y 348.163,Z 239.507,A -85,B 0,C 180,E1 15682.278,E2 15682.278} C_VEL
LIN {X 0,Y 344.882,Z 236.709,A -85,B 0,C 180,E1 15680.759,E2 15680.759} C_VEL
LIN {X 0,Y 342.763,Z 233.242,A -85,B 0,C 180,E1 15679.601,E2 15679.601} C_VEL
LIN {X 0,Y 339.343,Z 230.729,A -85,B 0,C 180,E1 15677.756,E2 15677.756} C_VEL
LIN {X 0,Y 337.495,Z 227.478,A -85,B 0,C 180,E1 15676.524,E2 15676.524} C_VEL
LIN {X 0,Y 336.219,Z 226.419,A -85,B 0,C 180,E1 15675.702,E2 15675.702} C_VEL
LIN {X 0,Y 332.951,Z 224.042,A -85,B 0,C 180,E1 15673.37,E2 15673.37} C_VEL
LIN {X 0,Y 331.258,Z 220.613,A -85,B 0,C 180,E1 15671.491,E2 15671.491} C_VEL
LIN {X 0,Y 331.136,Z 219.949,A -85,B 0,C 180,E1 15670.087,E2 15670.087} C_VEL
LIN {X 0,Y 331.132,Z 219.915,A -85,B 0,C 180,E1 15665.719,E2 15665.719} C_VEL
LIN {X 0,Y 331.144,Z 219.897,A -85,B 0,C 180,E1 15661.384,E2 15661.384} C_VEL
LIN {X 0,Y 331.154,Z 219.884,A -85,B 0,C 180,E1 15657.058,E2 15657.058} C_VEL
LIN {X 0,Y 331.145,Z 219.883,A -85,B 0,C 180,E1 15652.714,E2 15652.714} C_VEL
LIN {X 0,Y 331.185,Z 220.202,A -85,B 0,C 180,E1 15648.683,E2 15648.683} C_VEL
LIN {X 0,Y 331.546,Z 221.597,A -85,B 0,C 180,E1 15647.636,E2 15647.636} C_VEL
LIN {X 0,Y 333.53,Z 224.693,A -85,B 0,C 180,E1 15645.858,E2 15645.858} C_VEL
LIN {X 0,Y 337.381,Z 227.26,A -85,B 0,C 180,E1 15643.249,E2 15643.249} C_VEL
LIN {X 0,Y 339.279,Z 230.655,A -85,B 0,C 180,E1 15641.974,E2 15641.974} C_VEL
LIN {X 0,Y 342.528,Z 233.133,A -85,B 0,C 180,E1 15640.207,E2 15640.207} C_VEL
LIN {X 0,Y 343.208,Z 233.859,A -85,B 0,C 180,E1 15639.848,E2 15639.848} C_VEL
LIN {X 0,Y 345.523,Z 237.459,A -85,B 0,C 180,E1 15638.615,E2 15638.615} C_VEL
LIN {X 0,Y 348.589,Z 240.05,A -85,B 0,C 180,E1 15637.218,E2 15637.218} C_VEL
LIN {X 0,Y 351.494,Z 244.09,A -85,B 0,C 180,E1 15635.907,E2 15635.907} C_VEL
LIN {X 0,Y 353.737,Z 246.19,A -85,B 0,C 180,E1 15635.002,E2 15635.002} C_VEL
LIN {X 0,Y 357.13,Z 250.557,A -85,B 0,C 180,E1 15633.655,E2 15633.655} C_VEL
LIN {X 0,Y 358.715,Z 252.374,A -85,B 0,C 180,E1 15633.066,E2 15633.066} C_VEL
LIN {X 0,Y 363.603,Z 258.642,A -85,B 0,C 180,E1 15631.323,E2 15631.323} C_VEL
LIN {X 0,Y 368.338,Z 264.704,A -85,B 0,C 180,E1 15629.764,E2 15629.764} C_VEL
LIN {X 0,Y 375.036,Z 273.479,A -85,B 0,C 180,E1 15627.731,E2 15627.731} C_VEL
LIN {X 0,Y 390.245,Z 293.681,A -85,B 0,C 180,E1 15623.71,E2 15623.71} C_VEL
LIN {X 0,Y 405.989,Z 309.71,A -85,B 0,C 180,E1 15620.32,E2 15620.32} C_VEL
LIN {X 0,Y 416.463,Z 318.986,A -85,B 0,C 180,E1 15618.129,E2 15618.129} C_VEL
LIN {X 0,Y 425.591,Z 327.114,A -85,B 0,C 180,E1 15616.032,E2 15616.032} C_VEL
LIN {X 0,Y 434.18,Z 334.933,A -85,B 0,C 180,E1 15613.875,E2 15613.875} C_VEL
LIN {X 0,Y 441.973,Z 342.353,A -85,B 0,C 180,E1 15611.706,E2 15611.706} C_VEL
LIN {X 0,Y 449.765,Z 349.759,A -85,B 0,C 180,E1 15609.417,E2 15609.417} C_VEL
LIN {X 0,Y 457.666,Z 357.189,A -85,B 0,C 180,E1 15607.01,E2 15607.01} C_VEL
LIN {X 0,Y 466.041,Z 364.808,A -85,B 0,C 180,E1 15604.346,E2 15604.346} C_VEL
LIN {X 0,Y 470.386,Z 368.732,A -85,B 0,C 180,E1 15602.897,E2 15602.897} C_VEL
LIN {X 0,Y 476.511,Z 373.925,A -85,B 0,C 180,E1 15600.792,E2 15600.792} C_VEL
LIN {X 0,Y 482.601,Z 379.684,A -85,B 0,C 180,E1 15598.54,E2 15598.54} C_VEL
LIN {X 0,Y 487.204,Z 383.344,A -85,B 0,C 180,E1 15596.778,E2 15596.778} C_VEL
LIN {X 0,Y 492.527,Z 388.192,A -85,B 0,C 180,E1 15594.564,E2 15594.564} C_VEL
LIN {X 0,Y 496.642,Z 391.306,A -85,B 0,C 180,E1 15592.766,E2 15592.766} C_VEL
LIN {X 0,Y 501.189,Z 395.643,A -85,B 0,C 180,E1 15590.553,E2 15590.553} C_VEL
LIN {X 0,Y 505.555,Z 398.521,A -85,B 0,C 180,E1 15588.313,E2 15588.313} C_VEL
LIN {X 0,Y 509.621,Z 402.67,A -85,B 0,C 180,E1 15585.824,E2 15585.824} C_VEL
LIN {X 0,Y 513.001,Z 405.236,A -85,B 0,C 180,E1 15583.524,E2 15583.524} C_VEL
LIN {X 0,Y 516.11,Z 406.846,A -85,B 0,C 180,E1 15581.056,E2 15581.056} C_VEL
LIN {X 0,Y 517.115,Z 407.746,A -85,B 0,C 180,E1 15580.133,E2 15580.133} C_VEL
LIN {X 0,Y 519.061,Z 410.129,A -85,B 0,C 180,E1 15577.86,E2 15577.86} C_VEL
LIN {X 0,Y 520.535,Z 411.656,A -85,B 0,C 180,E1 15575.621,E2 15575.621} C_VEL
LIN {X 0,Y 521.714,Z 412.621,A -85,B 0,C 180,E1 15572.966,E2 15572.966} C_VEL
LIN {X 0,Y 522.139,Z 412.888,A -85,B 0,C 180,E1 15570.439,E2 15570.439} C_VEL
LIN {X 0,Y 521.92,Z 412.717,A -85,B 0,C 180,E1 15567.804,E2 15567.804} C_VEL
LIN {X 0,Y 521.063,Z 412.079,A -85,B 0,C 180,E1 15565.378,E2 15565.378} C_VEL
LIN {X 0,Y 519.48,Z 410.625,A -85,B 0,C 180,E1 15562.703,E2 15562.703} C_VEL
LIN {X 0,Y 517.529,Z 408.359,A -85,B 0,C 180,E1 15560.325,E2 15560.325} C_VEL
LIN {X 0,Y 516.243,Z 406.895,A -85,B 0,C 180,E1 15559.06,E2 15559.06} C_VEL
LIN {X 0,Y 513.35,Z 405.435,A -85,B 0,C 180,E1 15556.714,E2 15556.714} C_VEL
LIN {X 0,Y 509.875,Z 402.896,A -85,B 0,C 180,E1 15554.34,E2 15554.34} C_VEL
LIN {X 0,Y 506.34,Z 399.241,A -85,B 0,C 180,E1 15552.144,E2 15552.144} C_VEL
LIN {X 0,Y 501.452,Z 395.851,A -85,B 0,C 180,E1 15549.58,E2 15549.58} C_VEL
LIN {X 0,Y 496.868,Z 391.54,A -85,B 0,C 180,E1 15547.336,E2 15547.336} C_VEL
LIN {X 0,Y 494.199,Z 389.378,A -85,B 0,C 180,E1 15546.134,E2 15546.134} C_VEL
LIN {X 0,Y 488.891,Z 385.063,A -85,B 0,C 180,E1 15543.918,E2 15543.918} C_VEL
LIN {X 0,Y 485.256,Z 381.668,A -85,B 0,C 180,E1 15542.46,E2 15542.46} C_VEL
LIN {X 0,Y 479.575,Z 376.983,A -85,B 0,C 180,E1 15540.332,E2 15540.332} C_VEL
LIN {X 0,Y 475.696,Z 373.341,A -85,B 0,C 180,E1 15538.931,E2 15538.931} C_VEL
LIN {X 0,Y 469.456,Z 367.783,A -85,B 0,C 180,E1 15536.774,E2 15536.774} C_VEL
LIN {X 0,Y 461.266,Z 360.5,A -85,B 0,C 180,E1 15534.114,E2 15534.114} C_VEL
LIN {X 0,Y 456.577,Z 356.273,A -85,B 0,C 180,E1 15532.652,E2 15532.652} C_VEL
LIN {X 0,Y 448.868,Z 349.005,A -85,B 0,C 180,E1 15530.321,E2 15530.321} C_VEL
LIN {X 0,Y 439.716,Z 340.345,A -85,B 0,C 180,E1 15527.649,E2 15527.649} C_VEL
LIN {X 0,Y 432.633,Z 333.616,A -85,B 0,C 180,E1 15525.716,E2 15525.716} C_VEL
LIN {X 0,Y 424.559,Z 326.262,A -85,B 0,C 180,E1 15523.728,E2 15523.728} C_VEL
LIN {X 0,Y 415.387,Z 318.068,A -85,B 0,C 180,E1 15521.634,E2 15521.634} C_VEL
LIN {X 0,Y 404.275,Z 308.107,A -85,B 0,C 180,E1 15519.33,E2 15519.33} C_VEL
LIN {X 0,Y 389.193,Z 292.43,A -85,B 0,C 180,E1 15516.039,E2 15516.039} C_VEL
LIN {X 0,Y 377.743,Z 277.179,A -85,B 0,C 180,E1 15513.044,E2 15513.044} C_VEL
LIN {X 0,Y 369.336,Z 265.988,A -85,B 0,C 180,E1 15510.55,E2 15510.55} C_VEL
LIN {X 0,Y 365.51,Z 261.101,A -85,B 0,C 180,E1 15509.319,E2 15509.319} C_VEL
LIN {X 0,Y 361.529,Z 255.999,A -85,B 0,C 180,E1 15507.956,E2 15507.956} C_VEL
LIN {X 0,Y 357.533,Z 250.921,A -85,B 0,C 180,E1 15506.492,E2 15506.492} C_VEL
LIN {X 0,Y 354.002,Z 246.641,A -85,B 0,C 180,E1 15505.112,E2 15505.112} C_VEL
LIN {X 0,Y 352.993,Z 245.37,A -85,B 0,C 180,E1 15504.696,E2 15504.696} C_VEL
LIN {X 0,Y 349.65,Z 241.841,A -85,B 0,C 180,E1 15503.288,E2 15503.288} C_VEL
LIN {X 0,Y 348.08,Z 239.475,A -85,B 0,C 180,E1 15502.55,E2 15502.55} C_VEL
LIN {X 0,Y 344.733,Z 236.516,A -85,B 0,C 180,E1 15500.99,E2 15500.99} C_VEL
LIN {X 0,Y 342.849,Z 233.278,A -85,B 0,C 180,E1 15499.951,E2 15499.951} C_VEL
LIN {X 0,Y 339.552,Z 230.96,A -85,B 0,C 180,E1 15498.188,E2 15498.188} C_VEL
LIN {X 0,Y 337.606,Z 227.793,A -85,B 0,C 180,E1 15496.917,E2 15496.917} C_VEL
LIN {X 0,Y 336.818,Z 226.646,A -85,B 0,C 180,E1 15496.381,E2 15496.381} C_VEL
LIN {X 0,Y 333.105,Z 224.249,A -85,B 0,C 180,E1 15493.806,E2 15493.806} C_VEL
LIN {X 0,Y 331.268,Z 220.687,A -85,B 0,C 180,E1 15491.844,E2 15491.844} C_VEL
LIN {X 0,Y 331.146,Z 219.936,A -85,B 0,C 180,E1 15490.438,E2 15490.438} C_VEL
LIN {X 0,Y 331.126,Z 219.893,A -85,B 0,C 180,E1 15486.067,E2 15486.067} C_VEL
LIN {X 0,Y 331.128,Z 219.884,A -85,B 0,C 180,E1 15481.73,E2 15481.73} C_VEL
LIN {X 0,Y 331.135,Z 219.882,A -85,B 0,C 180,E1 15477.577,E2 15477.577} C_VEL
LIN {X 0,Y 331.161,Z 219.885,A -85,B 0,C 180,E1 15473.244,E2 15473.244} C_VEL
LIN {X 0,Y 331.009,Z 220.751,A -85,B 0,C 180,E1 15472.004,E2 15472.004} C_VEL
LIN {X 0,Y 330.399,Z 224.186,A -85,B 0,C 180,E1 15470.264,E2 15470.264} C_VEL
LIN {X 0,Y 330.533,Z 229.783,A -85,B 0,C 180,E1 15468.001,E2 15468.001} C_VEL
LIN {X 0,Y 331.085,Z 231.041,A -85,B 0,C 180,E1 15467.356,E2 15467.356} C_VEL
LIN {X 0,Y 333.772,Z 233.642,A -85,B 0,C 180,E1 15465.248,E2 15465.248} C_VEL
LIN {X 0,Y 335.769,Z 234.91,A -85,B 0,C 180,E1 15463.922,E2 15463.922} C_VEL
LIN {X 0,Y 337.831,Z 238.429,A -85,B 0,C 180,E1 15462.517,E2 15462.517} C_VEL
LIN {X 0,Y 341.366,Z 241.381,A -85,B 0,C 180,E1 15460.555,E2 15460.555} C_VEL
LIN {X 0,Y 343.991,Z 245.251,A -85,B 0,C 180,E1 15459.14,E2 15459.14} C_VEL
LIN {X 0,Y 346.584,Z 247.551,A -85,B 0,C 180,E1 15457.928,E2 15457.928} C_VEL
LIN {X 0,Y 349.717,Z 251.728,A -85,B 0,C 180,E1 15456.493,E2 15456.493} C_VEL
LIN {X 0,Y 351.731,Z 253.775,A -85,B 0,C 180,E1 15455.657,E2 15455.657} C_VEL
LIN {X 0,Y 355.287,Z 258.186,A -85,B 0,C 180,E1 15454.226,E2 15454.226} C_VEL
LIN {X 0,Y 361.055,Z 265.613,A -85,B 0,C 180,E1 15452.094,E2 15452.094} C_VEL
LIN {X 0,Y 368.126,Z 274.82,A -85,B 0,C 180,E1 15449.745,E2 15449.745} C_VEL
LIN {X 0,Y 376.793,Z 288.775,A -85,B 0,C 180,E1 15447.088,E2 15447.088} C_VEL
LIN {X 0,Y 384.982,Z 302.921,A -85,B 0,C 180,E1 15444.812,E2 15444.812} C_VEL
LIN {X 0,Y 393.243,Z 318.379,A -85,B 0,C 180,E1 15442.691,E2 15442.691} C_VEL
LIN {X 0,Y 400.426,Z 333.293,A -85,B 0,C 180,E1 15440.953,E2 15440.953} C_VEL
LIN {X 0,Y 389.438,Z 519.149,A -85,B 0,C 180,E1 15437.676,E2 15437.676} C_VEL
LIN {X 0,Y 387.525,Z 537.6,A -85,B 0,C 180,E1 15437.227,E2 15437.227} C_VEL
LIN {X 0,Y 384.237,Z 559.889,A -85,B 0,C 180,E1 15436.492,E2 15436.492} C_VEL
LIN {X 0,Y 380.217,Z 580.469,A -85,B 0,C 180,E1 15435.552,E2 15435.552} C_VEL
LIN {X 0,Y 376.206,Z 597.964,A -85,B 0,C 180,E1 15434.553,E2 15434.553} C_VEL
LIN {X 0,Y 372.059,Z 613.827,A -85,B 0,C 180,E1 15433.463,E2 15433.463} C_VEL
LIN {X 0,Y 367.584,Z 629.269,A -85,B 0,C 180,E1 15432.205,E2 15432.205} C_VEL
LIN {X 0,Y 362.823,Z 644.25,A -85,B 0,C 180,E1 15430.772,E2 15430.772} C_VEL
LIN {X 0,Y 357.44,Z 659.982,A -85,B 0,C 180,E1 15429,E2 15429} C_VEL
LIN {X 0,Y 350.801,Z 677.945,A -85,B 0,C 180,E1 15426.558,E2 15426.558} C_VEL
LIN {X 0,Y 345.522,Z 691.445,A -85,B 0,C 180,E1 15424.348,E2 15424.348} C_VEL
LIN {X 0,Y 340.748,Z 703.333,A -85,B 0,C 180,E1 15422.077,E2 15422.077} C_VEL
LIN {X 0,Y 336.49,Z 713.829,A -85,B 0,C 180,E1 15419.747,E2 15419.747} C_VEL
LIN {X 0,Y 332.502,Z 723.721,A -85,B 0,C 180,E1 15417.195,E2 15417.195} C_VEL
LIN {X 0,Y 328.916,Z 732.905,A -85,B 0,C 180,E1 15414.417,E2 15414.417} C_VEL
LIN {X 0,Y 325.523,Z 742.224,A -85,B 0,C 180,E1 15411.059,E2 15411.059} C_VEL
LIN {X 0,Y 322.708,Z 750.874,A -85,B 0,C 180,E1 15407.116,E2 15407.116} C_VEL
LIN {X 0,Y 321.187,Z 756.645,A -85,B 0,C 180,E1 15403.761,E2 15403.761} C_VEL
LIN {X 0,Y 320.405,Z 760.66,A -85,B 0,C 180,E1 15400.79,E2 15400.79} C_VEL
LIN {X 0,Y 320.035,Z 763.763,A -85,B 0,C 180,E1 15397.72,E2 15397.72} C_VEL
LIN {X 0,Y 319.938,Z 765.739,A -85,B 0,C 180,E1 15394.84,E2 15394.84} C_VEL
LIN {X 0,Y 319.963,Z 766.812,A -85,B 0,C 180,E1 15391.97,E2 15391.97} C_VEL
LIN {X 0,Y 319.971,Z 766.96,A -85,B 0,C 180,E1 15388.926,E2 15388.926} C_VEL
LIN {X 0,Y 319.945,Z 766.094,A -85,B 0,C 180,E1 15385.879,E2 15385.879} C_VEL
LIN {X 0,Y 319.998,Z 764.208,A -85,B 0,C 180,E1 15382.821,E2 15382.821} C_VEL
LIN {X 0,Y 320.312,Z 761.287,A -85,B 0,C 180,E1 15379.752,E2 15379.752} C_VEL
LIN {X 0,Y 321.04,Z 757.301,A -85,B 0,C 180,E1 15376.677,E2 15376.677} C_VEL
LIN {X 0,Y 322.316,Z 752.21,A -85,B 0,C 180,E1 15373.605,E2 15373.605} C_VEL
LIN {X 0,Y 324.23,Z 745.959,A -85,B 0,C 180,E1 15370.548,E2 15370.548} C_VEL
LIN {X 0,Y 326.835,Z 738.472,A -85,B 0,C 180,E1 15367.52,E2 15367.52} C_VEL
LIN {X 0,Y 330.861,Z 728.026,A -85,B 0,C 180,E1 15364.015,E2 15364.015} C_VEL
LIN {X 0,Y 335.645,Z 715.934,A -85,B 0,C 180,E1 15360.759,E2 15360.759} C_VEL
LIN {X 0,Y 340.106,Z 704.916,A -85,B 0,C 180,E1 15358.252,E2 15358.252} C_VEL
LIN {X 0,Y 344.809,Z 693.225,A -85,B 0,C 180,E1 15355.972,E2 15355.972} C_VEL
LIN {X 0,Y 349.628,Z 680.942,A -85,B 0,C 180,E1 15353.91,E2 15353.91} C_VEL
LIN {X 0,Y 354.668,Z 667.592,A -85,B 0,C 180,E1 15351.981,E2 15351.981} C_VEL
LIN {X 0,Y 360.541,Z 651.159,A -85,B 0,C 180,E1 15349.96,E2 15349.96} C_VEL
LIN {X 0,Y 366.856,Z 631.687,A -85,B 0,C 180,E1 15348.007,E2 15348.007} C_VEL
LIN {X 0,Y 371.552,Z 615.667,A -85,B 0,C 180,E1 15346.675,E2 15346.675} C_VEL
LIN {X 0,Y 375.683,Z 600.088,A -85,B 0,C 180,E1 15345.582,E2 15345.582} C_VEL
LIN {X 0,Y 379.406,Z 584.2,A -85,B 0,C 180,E1 15344.646,E2 15344.646} C_VEL
LIN {X 0,Y 382.699,Z 568.066,A -85,B 0,C 180,E1 15343.862,E2 15343.862} C_VEL
LIN {X 0,Y 385.62,Z 551.052,A -85,B 0,C 180,E1 15343.196,E2 15343.196} C_VEL
LIN {X 0,Y 388,Z 533.667,A -85,B 0,C 180,E1 15342.668,E2 15342.668} C_VEL
LIN {X 0,Y 389.762,Z 514.927,A -85,B 0,C 180,E1 15342.237,E2 15342.237} C_VEL
LIN {X 0,Y 400.351,Z 332.985,A -85,B 0,C 180,E1 15339.025,E2 15339.025} C_VEL
LIN {X 0,Y 391.337,Z 314.68,A -85,B 0,C 180,E1 15336.833,E2 15336.833} C_VEL
LIN {X 0,Y 382.071,Z 297.702,A -85,B 0,C 180,E1 15334.399,E2 15334.399} C_VEL
LIN {X 0,Y 373.566,Z 283.534,A -85,B 0,C 180,E1 15331.958,E2 15331.958} C_VEL
LIN {X 0,Y 367.129,Z 273.532,A -85,B 0,C 180,E1 15329.94,E2 15329.94} C_VEL
LIN {X 0,Y 359.428,Z 263.441,A -85,B 0,C 180,E1 15327.324,E2 15327.324} C_VEL
LIN {X 0,Y 355.089,Z 258.001,A -85,B 0,C 180,E1 15325.699,E2 15325.699} C_VEL
LIN {X 0,Y 351.47,Z 253.333,A -85,B 0,C 180,E1 15324.229,E2 15324.229} C_VEL
LIN {X 0,Y 347.385,Z 248.888,A -85,B 0,C 180,E1 15322.464,E2 15322.464} C_VEL
LIN {X 0,Y 346.001,Z 246.887,A -85,B 0,C 180,E1 15321.799,E2 15321.799} C_VEL
LIN {X 0,Y 342.674,Z 243.654,A -85,B 0,C 180,E1 15320.185,E2 15320.185} C_VEL
LIN {X 0,Y 340.882,Z 240.817,A -85,B 0,C 180,E1 15319.179,E2 15319.179} C_VEL
LIN {X 0,Y 337.436,Z 237.946,A -85,B 0,C 180,E1 15317.237,E2 15317.237} C_VEL
LIN {X 0,Y 335.536,Z 234.526,A -85,B 0,C 180,E1 15315.912,E2 15315.912} C_VEL
LIN {X 0,Y 331.77,Z 231.976,A -85,B 0,C 180,E1 15313.241,E2 15313.241} C_VEL
LIN {X 0,Y 329.301,Z 227.897,A -85,B 0,C 180,E1 15310.851,E2 15310.851} C_VEL
LIN {X 0,Y 323.907,Z 223.289,A -85,B 0,C 180,E1 15301.238,E2 15301.238} C_VEL
LIN {X 0,Y 323.953,Z 223.429,A -85,B 0,C 180,E1 15298.054,E2 15298.054} C_VEL
LIN {X 0,Y 329.603,Z 228.226,A -85,B 0,C 180,E1 15288.539,E2 15288.539} C_VEL
LIN {X 0,Y 332.135,Z 232.389,A -85,B 0,C 180,E1 15286.153,E2 15286.153} C_VEL
LIN {X 0,Y 335.77,Z 234.944,A -85,B 0,C 180,E1 15283.611,E2 15283.611} C_VEL
LIN {X 0,Y 337.771,Z 238.355,A -85,B 0,C 180,E1 15282.247,E2 15282.247} C_VEL
LIN {X 0,Y 341.329,Z 241.332,A -85,B 0,C 180,E1 15280.268,E2 15280.268} C_VEL
LIN {X 0,Y 343.92,Z 245.172,A -85,B 0,C 180,E1 15278.868,E2 15278.868} C_VEL
LIN {X 0,Y 346.676,Z 247.66,A -85,B 0,C 180,E1 15277.577,E2 15277.577} C_VEL
LIN {X 0,Y 350.001,Z 251.988,A -85,B 0,C 180,E1 15276.067,E2 15276.067} C_VEL
LIN {X 0,Y 351.74,Z 253.811,A -85,B 0,C 180,E1 15275.344,E2 15275.344} C_VEL
LIN {X 0,Y 355.4,Z 258.289,A -85,B 0,C 180,E1 15273.877,E2 15273.877} C_VEL
LIN {X 0,Y 361.169,Z 265.818,A -85,B 0,C 180,E1 15271.744,E2 15271.744} C_VEL
LIN {X 0,Y 368.262,Z 274.949,A -85,B 0,C 180,E1 15269.396,E2 15269.396} C_VEL
LIN {X 0,Y 378.427,Z 289.181,A -85,B 0,C 180,E1 15266.389,E2 15266.389} C_VEL
LIN {X 0,Y 389.201,Z 302.749,A -85,B 0,C 180,E1 15263.643,E2 15263.643} C_VEL
LIN {X 0,Y 403.997,Z 317.625,A -85,B 0,C 180,E1 15260.454,E2 15260.454} C_VEL
LIN {X 0,Y 415.249,Z 327.374,A -85,B 0,C 180,E1 15258.118,E2 15258.118} C_VEL
LIN {X 0,Y 423.284,Z 334.553,A -85,B 0,C 180,E1 15256.281,E2 15256.281} C_VEL
LIN {X 0,Y 431.493,Z 341.948,A -85,B 0,C 180,E1 15254.271,E2 15254.271} C_VEL
LIN {X 0,Y 439.634,Z 349.577,A -85,B 0,C 180,E1 15252.048,E2 15252.048} C_VEL
LIN {X 0,Y 447.704,Z 357.19,A -85,B 0,C 180,E1 15249.692,E2 15249.692} C_VEL
LIN {X 0,Y 455.855,Z 364.783,A -85,B 0,C 180,E1 15247.229,E2 15247.229} C_VEL
LIN {X 0,Y 464.125,Z 372.279,A -85,B 0,C 180,E1 15244.617,E2 15244.617} C_VEL
LIN {X 0,Y 468.743,Z 376.405,A -85,B 0,C 180,E1 15243.093,E2 15243.093} C_VEL
LIN {X 0,Y 474.81,Z 381.549,A -85,B 0,C 180,E1 15241.008,E2 15241.008} C_VEL
LIN {X 0,Y 481.167,Z 387.469,A -85,B 0,C 180,E1 15238.683,E2 15238.683} C_VEL
LIN {X 0,Y 485.783,Z 391.155,A -85,B 0,C 180,E1 15236.921,E2 15236.921} C_VEL
LIN {X 0,Y 491.056,Z 395.901,A -85,B 0,C 180,E1 15234.749,E2 15234.749} C_VEL
LIN {X 0,Y 495.396,Z 399.218,A -85,B 0,C 180,E1 15232.86,E2 15232.86} C_VEL
LIN {X 0,Y 500.082,Z 403.589,A -85,B 0,C 180,E1 15230.601,E2 15230.601} C_VEL
LIN {X 0,Y 504.529,Z 406.475,A -85,B 0,C 180,E1 15228.323,E2 15228.323} C_VEL
LIN {X 0,Y 508.464,Z 410.535,A -85,B 0,C 180,E1 15225.926,E2 15225.926} C_VEL
LIN {X 0,Y 511.8,Z 413.071,A -85,B 0,C 180,E1 15223.672,E2 15223.672} C_VEL
LIN {X 0,Y 514.968,Z 414.731,A -85,B 0,C 180,E1 15221.194,E2 15221.194} C_VEL
LIN {X 0,Y 516.009,Z 415.576,A -85,B 0,C 180,E1 15220.268,E2 15220.268} C_VEL
LIN {X 0,Y 517.988,Z 417.989,A -85,B 0,C 180,E1 15217.988,E2 15217.988} C_VEL
LIN {X 0,Y 519.51,Z 419.568,A -85,B 0,C 180,E1 15215.695,E2 15215.695} C_VEL
LIN {X 0,Y 520.736,Z 420.561,A -85,B 0,C 180,E1 15212.971,E2 15212.971} C_VEL
LIN {X 0,Y 521.153,Z 420.827,A -85,B 0,C 180,E1 15210.55,E2 15210.55} C_VEL
LIN {X 0,Y 520.941,Z 420.658,A -85,B 0,C 180,E1 15207.8,E2 15207.8} C_VEL
LIN {X 0,Y 520.083,Z 420.02,A -85,B 0,C 180,E1 15205.369,E2 15205.369} C_VEL
LIN {X 0,Y 518.486,Z 418.578,A -85,B 0,C 180,E1 15202.689,E2 15202.689} C_VEL
LIN {X 0,Y 516.446,Z 416.234,A -85,B 0,C 180,E1 15200.224,E2 15200.224} C_VEL
LIN {X 0,Y 515.233,Z 414.828,A -85,B 0,C 180,E1 15199.038,E2 15199.038} C_VEL
LIN {X 0,Y 512.318,Z 413.371,A -85,B 0,C 180,E1 15196.687,E2 15196.687} C_VEL
LIN {X 0,Y 508.859,Z 410.885,A -85,B 0,C 180,E1 15194.331,E2 15194.331} C_VEL
LIN {X 0,Y 505.228,Z 407.217,A -85,B 0,C 180,E1 15192.085,E2 15192.085} C_VEL
LIN {X 0,Y 502.464,Z 405.268,A -85,B 0,C 180,E1 15190.593,E2 15190.593} C_VEL
LIN {X 0,Y 497.862,Z 401.696,A -85,B 0,C 180,E1 15188.316,E2 15188.316} C_VEL
LIN {X 0,Y 493.681,Z 397.728,A -85,B 0,C 180,E1 15186.361,E2 15186.361} C_VEL
LIN {X 0,Y 488.269,Z 393.573,A -85,B 0,C 180,E1 15184.092,E2 15184.092} C_VEL
LIN {X 0,Y 483.637,Z 389.304,A -85,B 0,C 180,E1 15182.235,E2 15182.235} C_VEL
LIN {X 0,Y 477.743,Z 384.432,A -85,B 0,C 180,E1 15180.052,E2 15180.052} C_VEL
LIN {X 0,Y 473.595,Z 380.645,A -85,B 0,C 180,E1 15178.573,E2 15178.573} C_VEL
LIN {X 0,Y 467.004,Z 374.688,A -85,B 0,C 180,E1 15176.326,E2 15176.326} C_VEL
LIN {X 0,Y 459.569,Z 368.208,A -85,B 0,C 180,E1 15173.928,E2 15173.928} C_VEL
LIN {X 0,Y 454.313,Z 363.489,A -85,B 0,C 180,E1 15172.3,E2 15172.3} C_VEL
LIN {X 0,Y 446.356,Z 356.03,A -85,B 0,C 180,E1 15169.907,E2 15169.907} C_VEL
LIN {X 0,Y 438.015,Z 348.165,A -85,B 0,C 180,E1 15167.499,E2 15167.499} C_VEL
LIN {X 0,Y 430.491,Z 341.135,A -85,B 0,C 180,E1 15165.485,E2 15165.485} C_VEL
LIN {X 0,Y 421.588,Z 333.126,A -85,B 0,C 180,E1 15163.316,E2 15163.316} C_VEL
LIN {X 0,Y 412.615,Z 325.236,A -85,B 0,C 180,E1 15161.327,E2 15161.327} C_VEL
LIN {X 0,Y 402.691,Z 316.469,A -85,B 0,C 180,E1 15159.285,E2 15159.285} C_VEL
LIN {X 0,Y 386.954,Z 300.258,A -85,B 0,C 180,E1 15155.823,E2 15155.823} C_VEL
LIN {X 0,Y 374.983,Z 284.307,A -85,B 0,C 180,E1 15152.636,E2 15152.636} C_VEL
LIN {X 0,Y 367.039,Z 273.408,A -85,B 0,C 180,E1 15150.218,E2 15150.218} C_VEL
LIN {X 0,Y 361.993,Z 266.946,A -85,B 0,C 180,E1 15148.546,E2 15148.546} C_VEL
LIN {X 0,Y 358.926,Z 262.923,A -85,B 0,C 180,E1 15147.455,E2 15147.455} C_VEL
LIN {X 0,Y 355.201,Z 258.107,A -85,B 0,C 180,E1 15146.049,E2 15146.049} C_VEL
LIN {X 0,Y 351.565,Z 253.52,A -85,B 0,C 180,E1 15144.579,E2 15144.579} C_VEL
LIN {X 0,Y 347.318,Z 248.731,A -85,B 0,C 180,E1 15142.736,E2 15142.736} C_VEL
LIN {X 0,Y 346.098,Z 246.948,A -85,B 0,C 180,E1 15142.149,E2 15142.149} C_VEL
LIN {X 0,Y 342.756,Z 243.774,A -85,B 0,C 180,E1 15140.536,E2 15140.536} C_VEL
LIN {X 0,Y 340.967,Z 240.864,A -85,B 0,C 180,E1 15139.53,E2 15139.53} C_VEL
LIN {X 0,Y 337.638,Z 238.198,A -85,B 0,C 180,E1 15137.671,E2 15137.671} C_VEL
LIN {X 0,Y 335.348,Z 234.415,A -85,B 0,C 180,E1 15136.099,E2 15136.099} C_VEL
LIN {X 0,Y 331.721,Z 231.939,A -85,B 0,C 180,E1 15133.509,E2 15133.509} C_VEL
LIN {X 0,Y 329.344,Z 227.962,A -85,B 0,C 180,E1 15131.204,E2 15131.204} C_VEL
LIN {X 0,Y 323.909,Z 223.323,A -85,B 0,C 180,E1 15121.592,E2 15121.592} C_VEL
LIN {X 0,Y 323.972,Z 223.466,A -85,B 0,C 180,E1 15118.231,E2 15118.231} C_VEL
LIN {X 0,Y 329.643,Z 228.282,A -85,B 0,C 180,E1 15108.806,E2 15108.806} C_VEL
LIN {X 0,Y 331.085,Z 231.041,A -85,B 0,C 180,E1 15107.356,E2 15107.356} C_VEL
LIN {X 0,Y 332.13,Z 233.931,A -85,B 0,C 180,E1 15106.326,E2 15106.326} C_VEL
LIN {X 0,Y 334.242,Z 242.679,A -85,B 0,C 180,E1 15104.239,E2 15104.239} C_VEL
LIN {X 0,Y 334.684,Z 243.69,A -85,B 0,C 180,E1 15103.9,E2 15103.9} C_VEL
LIN {X 0,Y 337.278,Z 247.075,A -85,B 0,C 180,E1 15102.22,E2 15102.22} C_VEL
LIN {X 0,Y 339.602,Z 249,A -85,B 0,C 180,E1 15100.924,E2 15100.924} C_VEL
LIN {X 0,Y 342.394,Z 252.954,A -85,B 0,C 180,E1 15099.397,E2 15099.397} C_VEL
LIN {X 0,Y 344.689,Z 255.12,A -85,B 0,C 180,E1 15098.293,E2 15098.293} C_VEL
LIN {X 0,Y 348.228,Z 259.616,A -85,B 0,C 180,E1 15096.656,E2 15096.656} C_VEL
LIN {X 0,Y 349.836,Z 261.488,A -85,B 0,C 180,E1 15095.965,E2 15095.965} C_VEL
LIN {X 0,Y 354.489,Z 267.386,A -85,B 0,C 180,E1 15094.074,E2 15094.074} C_VEL
LIN {X 0,Y 358.841,Z 273.074,A -85,B 0,C 180,E1 15092.448,E2 15092.448} C_VEL
LIN {X 0,Y 365.167,Z 281.4,A -85,B 0,C 180,E1 15090.29,E2 15090.29} C_VEL
LIN {X 0,Y 373.56,Z 295.167,A -85,B 0,C 180,E1 15087.633,E2 15087.633} C_VEL
LIN {X 0,Y 381.544,Z 309.244,A -85,B 0,C 180,E1 15085.342,E2 15085.342} C_VEL
LIN {X 0,Y 389.483,Z 324.443,A -85,B 0,C 180,E1 15083.236,E2 15083.236} C_VEL
LIN {X 0,Y 395.201,Z 336.661,A -85,B 0,C 180,E1 15081.795,E2 15081.795} C_VEL
LIN {X 0,Y 384.083,Z 518.982,A -85,B 0,C 180,E1 15078.56,E2 15078.56} C_VEL
LIN {X 0,Y 382.125,Z 537.425,A -85,B 0,C 180,E1 15078.109,E2 15078.109} C_VEL
LIN {X 0,Y 378.754,Z 559.713,A -85,B 0,C 180,E1 15077.373,E2 15077.373} C_VEL
LIN {X 0,Y 374.628,Z 580.294,A -85,B 0,C 180,E1 15076.431,E2 15076.431} C_VEL
LIN {X 0,Y 370.507,Z 597.788,A -85,B 0,C 180,E1 15075.427,E2 15075.427} C_VEL
LIN {X 0,Y 366.242,Z 613.651,A -85,B 0,C 180,E1 15074.332,E2 15074.332} C_VEL
LIN {X 0,Y 361.635,Z 629.093,A -85,B 0,C 180,E1 15073.066,E2 15073.066} C_VEL
LIN {X 0,Y 356.729,Z 644.073,A -85,B 0,C 180,E1 15071.621,E2 15071.621} C_VEL
LIN {X 0,Y 351.168,Z 659.805,A -85,B 0,C 180,E1 15069.834,E2 15069.834} C_VEL
LIN {X 0,Y 344.09,Z 678.267,A -85,B 0,C 180,E1 15067.286,E2 15067.286} C_VEL
LIN {X 0,Y 338.818,Z 691.267,A -85,B 0,C 180,E1 15065.127,E2 15065.127} C_VEL
LIN {X 0,Y 333.856,Z 703.155,A -85,B 0,C 180,E1 15062.821,E2 15062.821} C_VEL
LIN {X 0,Y 329.419,Z 713.651,A -85,B 0,C 180,E1 15060.453,E2 15060.453} C_VEL
LIN {X 0,Y 325.249,Z 723.542,A -85,B 0,C 180,E1 15057.854,E2 15057.854} C_VEL
LIN {X 0,Y 321.484,Z 732.726,A -85,B 0,C 180,E1 15055.02,E2 15055.02} C_VEL
LIN {X 0,Y 317.91,Z 742.046,A -85,B 0,C 180,E1 15051.588,E2 15051.588} C_VEL
LIN {X 0,Y 314.924,Z 750.695,A -85,B 0,C 180,E1 15047.553,E2 15047.553} C_VEL
LIN {X 0,Y 313.34,Z 756.311,A -85,B 0,C 180,E1 15044.222,E2 15044.222} C_VEL
LIN {X 0,Y 312.457,Z 760.483,A -85,B 0,C 180,E1 15041.068,E2 15041.068} C_VEL
LIN {X 0,Y 312.047,Z 763.587,A -85,B 0,C 180,E1 15037.919,E2 15037.919} C_VEL
LIN {X 0,Y 311.939,Z 765.563,A -85,B 0,C 180,E1 15034.964,E2 15034.964} C_VEL
LIN {X 0,Y 311.964,Z 766.637,A -85,B 0,C 180,E1 15032.02,E2 15032.02} C_VEL
LIN {X 0,Y 311.972,Z 766.785,A -85,B 0,C 180,E1 15028.898,E2 15028.898} C_VEL
LIN {X 0,Y 311.945,Z 765.919,A -85,B 0,C 180,E1 15025.773,E2 15025.773} C_VEL
LIN {X 0,Y 312.008,Z 764.032,A -85,B 0,C 180,E1 15022.636,E2 15022.636} C_VEL
LIN {X 0,Y 312.351,Z 761.11,A -85,B 0,C 180,E1 15019.488,E2 15019.488} C_VEL
LIN {X 0,Y 313.141,Z 757.123,A -85,B 0,C 180,E1 15016.334,E2 15016.334} C_VEL
LIN {X 0,Y 314.508,Z 752.032,A -85,B 0,C 180,E1 15013.186,E2 15013.186} C_VEL
LIN {X 0,Y 316.541,Z 745.781,A -85,B 0,C 180,E1 15010.056,E2 15010.056} C_VEL
LIN {X 0,Y 319.295,Z 738.294,A -85,B 0,C 180,E1 15006.959,E2 15006.959} C_VEL
LIN {X 0,Y 323.528,Z 727.848,A -85,B 0,C 180,E1 15003.38,E2 15003.38} C_VEL
LIN {X 0,Y 328.536,Z 715.755,A -85,B 0,C 180,E1 15000.062,E2 15000.062} C_VEL
LIN {X 0,Y 333.301,Z 704.474,A -85,B 0,C 180,E1 14997.458,E2 14997.458} C_VEL
LIN {X 0,Y 338.08,Z 693.046,A -85,B 0,C 180,E1 14995.199,E2 14995.199} C_VEL
LIN {X 0,Y 343.08,Z 680.764,A -85,B 0,C 180,E1 14993.109,E2 14993.109} C_VEL
LIN {X 0,Y 348.299,Z 667.414,A -85,B 0,C 180,E1 14991.158,E2 14991.158} C_VEL
LIN {X 0,Y 354.368,Z 650.982,A -85,B 0,C 180,E1 14989.116,E2 14989.116} C_VEL
LIN {X 0,Y 360.884,Z 631.51,A -85,B 0,C 180,E1 14987.148,E2 14987.148} C_VEL
LIN {X 0,Y 365.719,Z 615.491,A -85,B 0,C 180,E1 14985.806,E2 14985.806} C_VEL
LIN {X 0,Y 369.967,Z 599.911,A -85,B 0,C 180,E1 14984.708,E2 14984.708} C_VEL
LIN {X 0,Y 373.977,Z 583.199,A -85,B 0,C 180,E1 14983.724,E2 14983.724} C_VEL
LIN {X 0,Y 377.372,Z 566.856,A -85,B 0,C 180,E1 14982.936,E2 14982.936} C_VEL
LIN {X 0,Y 380.353,Z 549.758,A -85,B 0,C 180,E1 14982.276,E2 14982.276} C_VEL
LIN {X 0,Y 382.882,Z 531.307,A -85,B 0,C 180,E1 14981.726,E2 14981.726} C_VEL
LIN {X 0,Y 385.01,Z 506.324,A -85,B 0,C 180,E1 14981.188,E2 14981.188} C_VEL
LIN {X 0,Y 395.135,Z 336.221,A -85,B 0,C 180,E1 14978.181,E2 14978.181} C_VEL
LIN {X 0,Y 386.671,Z 318.929,A -85,B 0,C 180,E1 14976.036,E2 14976.036} C_VEL
LIN {X 0,Y 378.035,Z 302.852,A -85,B 0,C 180,E1 14973.673,E2 14973.673} C_VEL
LIN {X 0,Y 370.169,Z 289.572,A -85,B 0,C 180,E1 14971.331,E2 14971.331} C_VEL
LIN {X 0,Y 364.295,Z 280.278,A -85,B 0,C 180,E1 14969.427,E2 14969.427} C_VEL
LIN {X 0,Y 356.84,Z 270.37,A -85,B 0,C 180,E1 14966.817,E2 14966.817} C_VEL
LIN {X 0,Y 352.587,Z 264.978,A -85,B 0,C 180,E1 14965.175,E2 14965.175} C_VEL
LIN {X 0,Y 348.591,Z 259.941,A -85,B 0,C 180,E1 14963.497,E2 14963.497} C_VEL
LIN {X 0,Y 344.924,Z 255.519,A -85,B 0,C 180,E1 14961.826,E2 14961.826} C_VEL
LIN {X 0,Y 343.869,Z 254.224,A -85,B 0,C 180,E1 14961.314,E2 14961.314} C_VEL
LIN {X 0,Y 340.575,Z 250.693,A -85,B 0,C 180,E1 14959.643,E2 14959.643} C_VEL
LIN {X 0,Y 339.328,Z 248.535,A -85,B 0,C 180,E1 14958.913,E2 14958.913} C_VEL
LIN {X 0,Y 335.811,Z 245.488,A -85,B 0,C 180,E1 14956.877,E2 14956.877} C_VEL
LIN {X 0,Y 333.813,Z 242.175,A -85,B 0,C 180,E1 14955.461,E2 14955.461} C_VEL
LIN {X 0,Y 330.294,Z 239.542,A -85,B 0,C 180,E1 14952.856,E2 14952.856} C_VEL
LIN {X 0,Y 328.161,Z 235.778,A -85,B 0,C 180,E1 14950.712,E2 14950.712} C_VEL
LIN {X 0,Y 322.915,Z 231.186,A -85,B 0,C 180,E1 14941.065,E2 14941.065} C_VEL
LIN {X 0,Y 323.004,Z 231.431,A -85,B 0,C 180,E1 14937.871,E2 14937.871} C_VEL
LIN {X 0,Y 328.372,Z 236.031,A -85,B 0,C 180,E1 14928.762,E2 14928.762} C_VEL
LIN {X 0,Y 330.646,Z 239.975,A -85,B 0,C 180,E1 14926.535,E2 14926.535} C_VEL
LIN {X 0,Y 334.175,Z 242.615,A -85,B 0,C 180,E1 14923.977,E2 14923.977} C_VEL
LIN {X 0,Y 336.534,Z 246.347,A -85,B 0,C 180,E1 14922.359,E2 14922.359} C_VEL
LIN {X 0,Y 339.608,Z 249.034,A -85,B 0,C 180,E1 14920.612,E2 14920.612} C_VEL
LIN {X 0,Y 342.484,Z 253.036,A -85,B 0,C 180,E1 14919.045,E2 14919.045} C_VEL
LIN {X 0,Y 344.783,Z 255.224,A -85,B 0,C 180,E1 14917.941,E2 14917.941} C_VEL
LIN {X 0,Y 348.332,Z 259.7,A -85,B 0,C 180,E1 14916.305,E2 14916.305} C_VEL
LIN {X 0,Y 349.847,Z 261.523,A -85,B 0,C 180,E1 14915.652,E2 14915.652} C_VEL
LIN {X 0,Y 354.313,Z 267.152,A -85,B 0,C 180,E1 14913.836,E2 14913.836} C_VEL
LIN {X 0,Y 358.956,Z 273.271,A -85,B 0,C 180,E1 14912.097,E2 14912.097} C_VEL
LIN {X 0,Y 365.518,Z 281.849,A -85,B 0,C 180,E1 14909.869,E2 14909.869} C_VEL
LIN {X 0,Y 375.405,Z 295.941,A -85,B 0,C 180,E1 14906.86,E2 14906.86} C_VEL
LIN {X 0,Y 386.566,Z 310.043,A -85,B 0,C 180,E1 14903.953,E2 14903.953} C_VEL
LIN {X 0,Y 400.968,Z 324.642,A -85,B 0,C 180,E1 14900.791,E2 14900.791} C_VEL
LIN {X 0,Y 411.512,Z 333.781,A -85,B 0,C 180,E1 14898.631,E2 14898.631} C_VEL
LIN {X 0,Y 421.296,Z 342.241,A -85,B 0,C 180,E1 14896.459,E2 14896.459} C_VEL
LIN {X 0,Y 428.59,Z 348.855,A -85,B 0,C 180,E1 14894.686,E2 14894.686} C_VEL
LIN {X 0,Y 436.951,Z 356.532,A -85,B 0,C 180,E1 14892.474,E2 14892.474} C_VEL
LIN {X 0,Y 445.956,Z 364.875,A -85,B 0,C 180,E1 14889.878,E2 14889.878} C_VEL
LIN {X 0,Y 453.821,Z 372.199,A -85,B 0,C 180,E1 14887.516,E2 14887.516} C_VEL
LIN {X 0,Y 462.331,Z 379.866,A -85,B 0,C 180,E1 14884.84,E2 14884.84} C_VEL
LIN {X 0,Y 467.498,Z 384.467,A -85,B 0,C 180,E1 14883.15,E2 14883.15} C_VEL
LIN {X 0,Y 475.197,Z 391.16,A -85,B 0,C 180,E1 14880.495,E2 14880.495} C_VEL
LIN {X 0,Y 481.068,Z 396.281,A -85,B 0,C 180,E1 14878.329,E2 14878.329} C_VEL
LIN {X 0,Y 484.353,Z 398.951,A -85,B 0,C 180,E1 14877.07,E2 14877.07} C_VEL
LIN {X 0,Y 489.748,Z 403.732,A -85,B 0,C 180,E1 14874.867,E2 14874.867} C_VEL
LIN {X 0,Y 493.929,Z 406.895,A -85,B 0,C 180,E1 14873.058,E2 14873.058} C_VEL
LIN {X 0,Y 498.718,Z 411.325,A -85,B 0,C 180,E1 14870.783,E2 14870.783} C_VEL
LIN {X 0,Y 503.099,Z 414.221,A -85,B 0,C 180,E1 14868.539,E2 14868.539} C_VEL
LIN {X 0,Y 507.329,Z 418.418,A -85,B 0,C 180,E1 14866.015,E2 14866.015} C_VEL
LIN {X 0,Y 510.77,Z 421.007,A -85,B 0,C 180,E1 14863.7,E2 14863.7} C_VEL
LIN {X 0,Y 513.958,Z 422.664,A -85,B 0,C 180,E1 14861.217,E2 14861.217} C_VEL
LIN {X 0,Y 514.995,Z 423.565,A -85,B 0,C 180,E1 14860.288,E2 14860.288} C_VEL
LIN {X 0,Y 517.072,Z 426.041,A -85,B 0,C 180,E1 14857.89,E2 14857.89} C_VEL
LIN {X 0,Y 518.564,Z 427.541,A -85,B 0,C 180,E1 14855.643,E2 14855.643} C_VEL
LIN {X 0,Y 519.758,Z 428.501,A -85,B 0,C 180,E1 14852.977,E2 14852.977} C_VEL
LIN {X 0,Y 520.178,Z 428.768,A -85,B 0,C 180,E1 14850.551,E2 14850.551} C_VEL
LIN {X 0,Y 519.962,Z 428.6,A -85,B 0,C 180,E1 14847.796,E2 14847.796} C_VEL
LIN {X 0,Y 519.102,Z 427.962,A -85,B 0,C 180,E1 14845.36,E2 14845.36} C_VEL
LIN {X 0,Y 517.49,Z 426.53,A -85,B 0,C 180,E1 14842.674,E2 14842.674} C_VEL
LIN {X 0,Y 515.409,Z 424.169,A -85,B 0,C 180,E1 14840.172,E2 14840.172} C_VEL
LIN {X 0,Y 514.091,Z 422.713,A -85,B 0,C 180,E1 14838.9,E2 14838.9} C_VEL
LIN {X 0,Y 510.94,Z 421.106,A -85,B 0,C 180,E1 14836.42,E2 14836.42} C_VEL
LIN {X 0,Y 507.515,Z 418.587,A -85,B 0,C 180,E1 14834.109,E2 14834.109} C_VEL
LIN {X 0,Y 503.716,Z 414.702,A -85,B 0,C 180,E1 14831.784,E2 14831.784} C_VEL
LIN {X 0,Y 498.847,Z 411.43,A -85,B 0,C 180,E1 14829.284,E2 14829.284} C_VEL
LIN {X 0,Y 494.083,Z 407.055,A -85,B 0,C 180,E1 14827.013,E2 14827.013} C_VEL
LIN {X 0,Y 490.794,Z 404.503,A -85,B 0,C 180,E1 14825.574,E2 14825.574} C_VEL
LIN {X 0,Y 485.332,Z 399.916,A -85,B 0,C 180,E1 14823.316,E2 14823.316} C_VEL
LIN {X 0,Y 481.927,Z 396.886,A -85,B 0,C 180,E1 14821.985,E2 14821.985} C_VEL
LIN {X 0,Y 476.212,Z 392.173,A -85,B 0,C 180,E1 14819.884,E2 14819.884} C_VEL
LIN {X 0,Y 471.734,Z 388.119,A -85,B 0,C 180,E1 14818.292,E2 14818.292} C_VEL
LIN {X 0,Y 465.146,Z 382.194,A -85,B 0,C 180,E1 14816.074,E2 14816.074} C_VEL
LIN {X 0,Y 457.543,Z 375.598,A -85,B 0,C 180,E1 14813.64,E2 14813.64} C_VEL
LIN {X 0,Y 448.396,Z 367.231,A -85,B 0,C 180,E1 14810.847,E2 14810.847} C_VEL
LIN {X 0,Y 439.413,Z 358.754,A -85,B 0,C 180,E1 14808.216,E2 14808.216} C_VEL
LIN {X 0,Y 431.779,Z 351.682,A -85,B 0,C 180,E1 14806.119,E2 14806.119} C_VEL
LIN {X 0,Y 423.21,Z 344.025,A -85,B 0,C 180,E1 14803.997,E2 14803.997} C_VEL
LIN {X 0,Y 414.433,Z 336.224,A -85,B 0,C 180,E1 14801.988,E2 14801.988} C_VEL
LIN {X 0,Y 405.034,Z 328.047,A -85,B 0,C 180,E1 14800.022,E2 14800.022} C_VEL
LIN {X 0,Y 395.557,Z 319.413,A -85,B 0,C 180,E1 14798.082,E2 14798.082} C_VEL
LIN {X 0,Y 383.048,Z 306.049,A -85,B 0,C 180,E1 14795.186,E2 14795.186} C_VEL
LIN {X 0,Y 371.562,Z 290.333,A -85,B 0,C 180,E1 14792.015,E2 14792.015} C_VEL
LIN {X 0,Y 363.453,Z 279.188,A -85,B 0,C 180,E1 14789.456,E2 14789.456} C_VEL
LIN {X 0,Y 356.654,Z 270.18,A -85,B 0,C 180,E1 14787.057,E2 14787.057} C_VEL
LIN {X 0,Y 352.698,Z 265.093,A -85,B 0,C 180,E1 14785.526,E2 14785.526} C_VEL
LIN {X 0,Y 348.514,Z 259.862,A -85,B 0,C 180,E1 14783.772,E2 14783.772} C_VEL
LIN {X 0,Y 344.939,Z 255.489,A -85,B 0,C 180,E1 14782.138,E2 14782.138} C_VEL
LIN {X 0,Y 343.796,Z 254.162,A -85,B 0,C 180,E1 14781.587,E2 14781.587} C_VEL
LIN {X 0,Y 340.44,Z 250.49,A -85,B 0,C 180,E1 14779.875,E2 14779.875} C_VEL
LIN {X 0,Y 339.106,Z 248.423,A -85,B 0,C 180,E1 14779.105,E2 14779.105} C_VEL
LIN {X 0,Y 335.755,Z 245.413,A -85,B 0,C 180,E1 14777.147,E2 14777.147} C_VEL
LIN {X 0,Y 333.885,Z 242.189,A -85,B 0,C 180,E1 14775.814,E2 14775.814} C_VEL
LIN {X 0,Y 330.345,Z 239.629,A -85,B 0,C 180,E1 14773.21,E2 14773.21} C_VEL
LIN {X 0,Y 328.035,Z 235.689,A -85,B 0,C 180,E1 14770.893,E2 14770.893} C_VEL
LIN {X 0,Y 322.916,Z 231.222,A -85,B 0,C 180,E1 14761.419,E2 14761.419} C_VEL
LIN {X 0,Y 322.996,Z 231.42,A -85,B 0,C 180,E1 14758.226,E2 14758.226} C_VEL
LIN {X 0,Y 328.409,Z 236.098,A -85,B 0,C 180,E1 14749.03,E2 14749.03} C_VEL
LIN {X 0,Y 330.694,Z 240.013,A -85,B 0,C 180,E1 14746.804,E2 14746.804} C_VEL
LIN {X 0,Y 334.172,Z 242.586,A -85,B 0,C 180,E1 14744.289,E2 14744.289} C_VEL
LIN {X 0,Y 334.684,Z 243.69,A -85,B 0,C 180,E1 14743.9,E2 14743.9} C_VEL
LIN {X 0,Y 335.869,Z 247.381,A -85,B 0,C 180,E1 14742.956,E2 14742.956} C_VEL
LIN {X 0,Y 337.956,Z 256.392,A -85,B 0,C 180,E1 14741.26,E2 14741.26} C_VEL
LIN {X 0,Y 338.817,Z 258.21,A -85,B 0,C 180,E1 14740.725,E2 14740.725} C_VEL
LIN {X 0,Y 342.261,Z 261.913,A -85,B 0,C 180,E1 14738.94,E2 14738.94} C_VEL
LIN {X 0,Y 346.386,Z 267.158,A -85,B 0,C 180,E1 14736.974,E2 14736.974} C_VEL
LIN {X 0,Y 352.095,Z 274.425,A -85,B 0,C 180,E1 14734.555,E2 14734.555} C_VEL
LIN {X 0,Y 356.844,Z 280.786,A -85,B 0,C 180,E1 14732.733,E2 14732.733} C_VEL
LIN {X 0,Y 362.55,Z 288.536,A -85,B 0,C 180,E1 14730.735,E2 14730.735} C_VEL
LIN {X 0,Y 370.473,Z 301.751,A -85,B 0,C 180,E1 14728.153,E2 14728.153} C_VEL
LIN {X 0,Y 378.555,Z 316.326,A -85,B 0,C 180,E1 14725.764,E2 14725.764} C_VEL
LIN {X 0,Y 386.954,Z 332.987,A -85,B 0,C 180,E1 14723.477,E2 14723.477} C_VEL
LIN {X 0,Y 390.066,Z 339.994,A -85,B 0,C 180,E1 14722.659,E2 14722.659} C_VEL
LIN {X 0,Y 378.823,Z 518.815,A -85,B 0,C 180,E1 14719.47,E2 14719.47} C_VEL
LIN {X 0,Y 376.799,Z 537.397,A -85,B 0,C 180,E1 14719.013,E2 14719.013} C_VEL
LIN {X 0,Y 373.364,Z 559.538,A -85,B 0,C 180,E1 14718.28,E2 14718.28} C_VEL
LIN {X 0,Y 369.129,Z 580.118,A -85,B 0,C 180,E1 14717.335,E2 14717.335} C_VEL
LIN {X 0,Y 364.89,Z 597.641,A -85,B 0,C 180,E1 14716.327,E2 14716.327} C_VEL
LIN {X 0,Y 360.515,Z 613.474,A -85,B 0,C 180,E1 14715.228,E2 14715.228} C_VEL
LIN {X 0,Y 355.771,Z 628.916,A -85,B 0,C 180,E1 14713.955,E2 14713.955} C_VEL
LIN {X 0,Y 350.716,Z 643.896,A -85,B 0,C 180,E1 14712.5,E2 14712.5} C_VEL
LIN {X 0,Y 344.972,Z 659.627,A -85,B 0,C 180,E1 14710.697,E2 14710.697} C_VEL
LIN {X 0,Y 337.65,Z 678.089,A -85,B 0,C 180,E1 14708.123,E2 14708.123} C_VEL
LIN {X 0,Y 332.154,Z 691.148,A -85,B 0,C 180,E1 14705.925,E2 14705.925} C_VEL
LIN {X 0,Y 327.023,Z 702.977,A -85,B 0,C 180,E1 14703.596,E2 14703.596} C_VEL
LIN {X 0,Y 322.184,Z 713.963,A -85,B 0,C 180,E1 14701.067,E2 14701.067} C_VEL
LIN {X 0,Y 317.774,Z 723.982,A -85,B 0,C 180,E1 14698.363,E2 14698.363} C_VEL
LIN {X 0,Y 313.65,Z 733.631,A -85,B 0,C 180,E1 14695.285,E2 14695.285} C_VEL
LIN {X 0,Y 309.335,Z 744.402,A -85,B 0,C 180,E1 14691.023,E2 14691.023} C_VEL
LIN {X 0,Y 306.932,Z 751.186,A -85,B 0,C 180,E1 14687.633,E2 14687.633} C_VEL
LIN {X 0,Y 305.393,Z 756.405,A -85,B 0,C 180,E1 14684.406,E2 14684.406} C_VEL
LIN {X 0,Y 304.472,Z 760.515,A -85,B 0,C 180,E1 14681.171,E2 14681.171} C_VEL
LIN {X 0,Y 304.048,Z 763.559,A -85,B 0,C 180,E1 14677.938,E2 14677.938} C_VEL
LIN {X 0,Y 303.94,Z 765.477,A -85,B 0,C 180,E1 14674.906,E2 14674.906} C_VEL
LIN {X 0,Y 303.967,Z 766.492,A -85,B 0,C 180,E1 14671.885,E2 14671.885} C_VEL
LIN {X 0,Y 303.973,Z 766.61,A -85,B 0,C 180,E1 14668.869,E2 14668.869} C_VEL
LIN {X 0,Y 303.944,Z 765.744,A -85,B 0,C 180,E1 14665.661,E2 14665.661} C_VEL
LIN {X 0,Y 304.022,Z 763.856,A -85,B 0,C 180,E1 14662.442,E2 14662.442} C_VEL
LIN {X 0,Y 304.408,Z 760.871,A -85,B 0,C 180,E1 14659.153,E2 14659.153} C_VEL
LIN {X 0,Y 305.253,Z 756.946,A -85,B 0,C 180,E1 14655.974,E2 14655.974} C_VEL
LIN {X 0,Y 306.715,Z 751.854,A -85,B 0,C 180,E1 14652.745,E2 14652.745} C_VEL
LIN {X 0,Y 308.877,Z 745.602,A -85,B 0,C 180,E1 14649.539,E2 14649.539} C_VEL
LIN {X 0,Y 311.787,Z 738.115,A -85,B 0,C 180,E1 14646.371,E2 14646.371} C_VEL
LIN {X 0,Y 316.322,Z 727.472,A -85,B 0,C 180,E1 14642.654,E2 14642.654} C_VEL
LIN {X 0,Y 321.479,Z 715.577,A -85,B 0,C 180,E1 14639.335,E2 14639.335} C_VEL
LIN {X 0,Y 326.332,Z 704.559,A -85,B 0,C 180,E1 14636.744,E2 14636.744} C_VEL
LIN {X 0,Y 331.035,Z 693.758,A -85,B 0,C 180,E1 14634.56,E2 14634.56} C_VEL
LIN {X 0,Y 336.188,Z 681.585,A -85,B 0,C 180,E1 14632.437,E2 14632.437} C_VEL
LIN {X 0,Y 341.337,Z 668.918,A -85,B 0,C 180,E1 14630.537,E2 14630.537} C_VEL
LIN {X 0,Y 346.604,Z 655.216,A -85,B 0,C 180,E1 14628.769,E2 14628.769} C_VEL
LIN {X 0,Y 351.942,Z 640.398,A -85,B 0,C 180,E1 14627.138,E2 14627.138} C_VEL
LIN {X 0,Y 357.866,Z 622.47,A -85,B 0,C 180,E1 14625.476,E2 14625.476} C_VEL
LIN {X 0,Y 363.794,Z 601.86,A -85,B 0,C 180,E1 14623.945,E2 14623.945} C_VEL
LIN {X 0,Y 367.991,Z 585.092,A -85,B 0,C 180,E1 14622.931,E2 14622.931} C_VEL
LIN {X 0,Y 371.597,Z 568.458,A -85,B 0,C 180,E1 14622.108,E2 14622.108} C_VEL
LIN {X 0,Y 374.72,Z 551.297,A -85,B 0,C 180,E1 14621.428,E2 14621.428} C_VEL
LIN {X 0,Y 377.232,Z 533.977,A -85,B 0,C 180,E1 14620.895,E2 14620.895} C_VEL
LIN {X 0,Y 379.052,Z 515.992,A -85,B 0,C 180,E1 14620.472,E2 14620.472} C_VEL
LIN {X 0,Y 390.033,Z 339.573,A -85,B 0,C 180,E1 14617.322,E2 14617.322} C_VEL
LIN {X 0,Y 382.145,Z 323.261,A -85,B 0,C 180,E1 14615.236,E2 14615.236} C_VEL
LIN {X 0,Y 373.656,Z 307.309,A -85,B 0,C 180,E1 14612.812,E2 14612.812} C_VEL
LIN {X 0,Y 366.818,Z 295.605,A -85,B 0,C 180,E1 14610.692,E2 14610.692} C_VEL
LIN {X 0,Y 361.385,Z 286.884,A -85,B 0,C 180,E1 14608.869,E2 14608.869} C_VEL
LIN {X 0,Y 354.184,Z 277.172,A -85,B 0,C 180,E1 14606.265,E2 14606.265} C_VEL
LIN {X 0,Y 350.212,Z 272.038,A -85,B 0,C 180,E1 14604.681,E2 14604.681} C_VEL
LIN {X 0,Y 346.386,Z 267.158,A -85,B 0,C 180,E1 14603.026,E2 14603.026} C_VEL
LIN {X 0,Y 342.659,Z 262.402,A -85,B 0,C 180,E1 14601.258,E2 14601.258} C_VEL
LIN {X 0,Y 338.647,Z 257.948,A -85,B 0,C 180,E1 14599.177,E2 14599.177} C_VEL
LIN {X 0,Y 337.483,Z 256.065,A -85,B 0,C 180,E1 14598.483,E2 14598.483} C_VEL
LIN {X 0,Y 334.077,Z 252.86,A -85,B 0,C 180,E1 14596.43,E2 14596.43} C_VEL
LIN {X 0,Y 332.361,Z 249.935,A -85,B 0,C 180,E1 14595.173,E2 14595.173} C_VEL
LIN {X 0,Y 328.929,Z 247.23,A -85,B 0,C 180,E1 14592.553,E2 14592.553} C_VEL
LIN {X 0,Y 326.856,Z 243.515,A -85,B 0,C 180,E1 14590.398,E2 14590.398} C_VEL
LIN {X 0,Y 321.924,Z 239.094,A -85,B 0,C 180,E1 14580.89,E2 14580.89} C_VEL
LIN {X 0,Y 322.058,Z 239.434,A -85,B 0,C 180,E1 14577.687,E2 14577.687} C_VEL
LIN {X 0,Y 327.142,Z 243.873,A -85,B 0,C 180,E1 14568.987,E2 14568.987} C_VEL
LIN {X 0,Y 329.272,Z 247.668,A -85,B 0,C 180,E1 14566.835,E2 14566.835} C_VEL
LIN {X 0,Y 332.65,Z 250.366,A -85,B 0,C 180,E1 14564.305,E2 14564.305} C_VEL
LIN {X 0,Y 335.169,Z 254.18,A -85,B 0,C 180,E1 14562.553,E2 14562.553} C_VEL
LIN {X 0,Y 337.904,Z 256.687,A -85,B 0,C 180,E1 14560.959,E2 14560.959} C_VEL
LIN {X 0,Y 341.053,Z 260.886,A -85,B 0,C 180,E1 14559.222,E2 14559.222} C_VEL
LIN {X 0,Y 342.906,Z 262.763,A -85,B 0,C 180,E1 14558.309,E2 14558.309} C_VEL
LIN {X 0,Y 346.67,Z 267.406,A -85,B 0,C 180,E1 14556.545,E2 14556.545} C_VEL
LIN {X 0,Y 352.186,Z 274.584,A -85,B 0,C 180,E1 14554.209,E2 14554.209} C_VEL
LIN {X 0,Y 356.86,Z 280.843,A -85,B 0,C 180,E1 14552.418,E2 14552.418} C_VEL
LIN {X 0,Y 363.118,Z 289.233,A -85,B 0,C 180,E1 14550.242,E2 14550.242} C_VEL
LIN {X 0,Y 372.41,Z 302.695,A -85,B 0,C 180,E1 14547.339,E2 14547.339} C_VEL
LIN {X 0,Y 383.548,Z 316.922,A -85,B 0,C 180,E1 14544.362,E2 14544.362} C_VEL
LIN {X 0,Y 397.801,Z 331.532,A -85,B 0,C 180,E1 14541.161,E2 14541.161} C_VEL
LIN {X 0,Y 409.002,Z 341.172,A -85,B 0,C 180,E1 14538.881,E2 14538.881} C_VEL
LIN {X 0,Y 418.835,Z 349.546,A -85,B 0,C 180,E1 14536.752,E2 14536.752} C_VEL
LIN {X 0,Y 426.751,Z 356.623,A -85,B 0,C 180,E1 14534.842,E2 14534.842} C_VEL
LIN {X 0,Y 434.641,Z 363.821,A -85,B 0,C 180,E1 14532.789,E2 14532.789} C_VEL
LIN {X 0,Y 443.529,Z 372.007,A -85,B 0,C 180,E1 14530.26,E2 14530.26} C_VEL
LIN {X 0,Y 451.754,Z 379.616,A -85,B 0,C 180,E1 14527.799,E2 14527.799} C_VEL
LIN {X 0,Y 460.289,Z 387.256,A -85,B 0,C 180,E1 14525.14,E2 14525.14} C_VEL
LIN {X 0,Y 464.986,Z 391.372,A -85,B 0,C 180,E1 14523.614,E2 14523.614} C_VEL
LIN {X 0,Y 471.533,Z 396.871,A -85,B 0,C 180,E1 14521.405,E2 14521.405} C_VEL
LIN {X 0,Y 478.092,Z 402.871,A -85,B 0,C 180,E1 14519.048,E2 14519.048} C_VEL
LIN {X 0,Y 482.716,Z 406.54,A -85,B 0,C 180,E1 14517.299,E2 14517.299} C_VEL
LIN {X 0,Y 488.228,Z 411.396,A -85,B 0,C 180,E1 14515.08,E2 14515.08} C_VEL
LIN {X 0,Y 492.609,Z 414.73,A -85,B 0,C 180,E1 14513.186,E2 14513.186} C_VEL
LIN {X 0,Y 497.354,Z 419.061,A -85,B 0,C 180,E1 14510.965,E2 14510.965} C_VEL
LIN {X 0,Y 502.012,Z 422.144,A -85,B 0,C 180,E1 14508.581,E2 14508.581} C_VEL
LIN {X 0,Y 506.084,Z 426.205,A -85,B 0,C 180,E1 14506.173,E2 14506.173} C_VEL
LIN {X 0,Y 509.646,Z 428.888,A -85,B 0,C 180,E1 14503.794,E2 14503.794} C_VEL
LIN {X 0,Y 512.949,Z 430.598,A -85,B 0,C 180,E1 14501.239,E2 14501.239} C_VEL
LIN {X 0,Y 514.096,Z 431.706,A -85,B 0,C 180,E1 14500.193,E2 14500.193} C_VEL
LIN {X 0,Y 516.156,Z 434.099,A -85,B 0,C 180,E1 14497.792,E2 14497.792} C_VEL
LIN {X 0,Y 517.65,Z 435.536,A -85,B 0,C 180,E1 14495.542,E2 14495.542} C_VEL
LIN {X 0,Y 518.803,Z 436.457,A -85,B 0,C 180,E1 14492.872,E2 14492.872} C_VEL
LIN {X 0,Y 519.214,Z 436.709,A -85,B 0,C 180,E1 14490.441,E2 14490.441} C_VEL
LIN {X 0,Y 518.983,Z 436.541,A -85,B 0,C 180,E1 14487.792,E2 14487.792} C_VEL
LIN {X 0,Y 518.122,Z 435.903,A -85,B 0,C 180,E1 14485.352,E2 14485.352} C_VEL
LIN {X 0,Y 516.495,Z 434.482,A -85,B 0,C 180,E1 14482.66,E2 14482.66} C_VEL
LIN {X 0,Y 514.403,Z 432.143,A -85,B 0,C 180,E1 14480.152,E2 14480.152} C_VEL
LIN {X 0,Y 513.082,Z 430.647,A -85,B 0,C 180,E1 14478.878,E2 14478.878} C_VEL
LIN {X 0,Y 509.91,Z 429.043,A -85,B 0,C 180,E1 14476.392,E2 14476.392} C_VEL
LIN {X 0,Y 506.433,Z 426.517,A -85,B 0,C 180,E1 14474.055,E2 14474.055} C_VEL
LIN {X 0,Y 502.466,Z 422.547,A -85,B 0,C 180,E1 14471.662,E2 14471.662} C_VEL
LIN {X 0,Y 497.56,Z 419.228,A -85,B 0,C 180,E1 14469.141,E2 14469.141} C_VEL
LIN {X 0,Y 492.662,Z 414.784,A -85,B 0,C 180,E1 14466.838,E2 14466.838} C_VEL
LIN {X 0,Y 488.912,Z 411.92,A -85,B 0,C 180,E1 14465.216,E2 14465.216} C_VEL
LIN {X 0,Y 483.295,Z 407.117,A -85,B 0,C 180,E1 14462.929,E2 14462.929} C_VEL
LIN {X 0,Y 480.201,Z 404.467,A -85,B 0,C 180,E1 14461.738,E2 14461.738} C_VEL
LIN {X 0,Y 474.194,Z 399.433,A -85,B 0,C 180,E1 14459.53,E2 14459.53} C_VEL
LIN {X 0,Y 469.6,Z 395.403,A -85,B 0,C 180,E1 14457.934,E2 14457.934} C_VEL
LIN {X 0,Y 463.036,Z 389.43,A -85,B 0,C 180,E1 14455.732,E2 14455.732} C_VEL
LIN {X 0,Y 455.83,Z 383.309,A -85,B 0,C 180,E1 14453.455,E2 14453.455} C_VEL
LIN {X 0,Y 449.211,Z 377.417,A -85,B 0,C 180,E1 14451.43,E2 14451.43} C_VEL
LIN {X 0,Y 442.161,Z 370.857,A -85,B 0,C 180,E1 14449.349,E2 14449.349} C_VEL
LIN {X 0,Y 433.488,Z 362.803,A -85,B 0,C 180,E1 14446.89,E2 14446.89} C_VEL
LIN {X 0,Y 424.482,Z 354.694,A -85,B 0,C 180,E1 14444.584,E2 14444.584} C_VEL
LIN {X 0,Y 415.984,Z 347.273,A -85,B 0,C 180,E1 14442.628,E2 14442.628} C_VEL
LIN {X 0,Y 406.072,Z 338.725,A -85,B 0,C 180,E1 14440.5,E2 14440.5} C_VEL
LIN {X 0,Y 392.581,Z 326.442,A -85,B 0,C 180,E1 14437.728,E2 14437.728} C_VEL
LIN {X 0,Y 379.945,Z 312.778,A -85,B 0,C 180,E1 14434.733,E2 14434.733} C_VEL
LIN {X 0,Y 368.518,Z 296.908,A -85,B 0,C 180,E1 14431.487,E2 14431.487} C_VEL
LIN {X 0,Y 360.458,Z 285.635,A -85,B 0,C 180,E1 14428.86,E2 14428.86} C_VEL
LIN {X 0,Y 353.808,Z 276.746,A -85,B 0,C 180,E1 14426.43,E2 14426.43} C_VEL
LIN {X 0,Y 350.228,Z 272.059,A -85,B 0,C 180,E1 14424.995,E2 14424.995} C_VEL
LIN {X 0,Y 346.313,Z 267.076,A -85,B 0,C 180,E1 14423.3,E2 14423.3} C_VEL
LIN {X 0,Y 342.676,Z 262.372,A -85,B 0,C 180,E1 14421.571,E2 14421.571} C_VEL
LIN {X 0,Y 338.656,Z 257.969,A -85,B 0,C 180,E1 14419.49,E2 14419.49} C_VEL
LIN {X 0,Y 337.566,Z 256.135,A -85,B 0,C 180,E1 14418.836,E2 14418.836} C_VEL
LIN {X 0,Y 334.023,Z 252.786,A -85,B 0,C 180,E1 14416.701,E2 14416.701} C_VEL
LIN {X 0,Y 332.432,Z 249.954,A -85,B 0,C 180,E1 14415.527,E2 14415.527} C_VEL
LIN {X 0,Y 328.884,Z 247.197,A -85,B 0,C 180,E1 14412.823,E2 14412.823} C_VEL
LIN {X 0,Y 326.899,Z 243.572,A -85,B 0,C 180,E1 14410.753,E2 14410.753} C_VEL
LIN {X 0,Y 321.926,Z 239.121,A -85,B 0,C 180,E1 14401.246,E2 14401.246} C_VEL
LIN {X 0,Y 322.048,Z 239.431,A -85,B 0,C 180,E1 14398.043,E2 14398.043} C_VEL
LIN {X 0,Y 327.101,Z 243.788,A -85,B 0,C 180,E1 14389.342,E2 14389.342} C_VEL
LIN {X 0,Y 329.318,Z 247.704,A -85,B 0,C 180,E1 14387.105,E2 14387.105} C_VEL
LIN {X 0,Y 332.646,Z 250.339,A -85,B 0,C 180,E1 14384.617,E2 14384.617} C_VEL
LIN {X 0,Y 335.227,Z 254.242,A -85,B 0,C 180,E1 14382.825,E2 14382.825} C_VEL
LIN {X 0,Y 337.897,Z 256.656,A -85,B 0,C 180,E1 14381.272,E2 14381.272} C_VEL
LIN {X 0,Y 338.817,Z 258.21,A -85,B 0,C 180,E1 14380.725,E2 14380.725} C_VEL
LIN {X 0,Y 340.683,Z 262.049,A -85,B 0,C 180,E1 14379.627,E2 14379.627} C_VEL
LIN {X 0,Y 345.675,Z 275.832,A -85,B 0,C 180,E1 14376.802,E2 14376.802} C_VEL
LIN {X 0,Y 347.346,Z 278.475,A -85,B 0,C 180,E1 14376.04,E2 14376.04} C_VEL
LIN {X 0,Y 350.059,Z 281.958,A -85,B 0,C 180,E1 14374.902,E2 14374.902} C_VEL
LIN {X 0,Y 356.676,Z 290.831,A -85,B 0,C 180,E1 14372.357,E2 14372.357} C_VEL
LIN {X 0,Y 360.571,Z 296.724,A -85,B 0,C 180,E1 14370.968,E2 14370.968} C_VEL
LIN {X 0,Y 367.319,Z 308.161,A -85,B 0,C 180,E1 14368.713,E2 14368.713} C_VEL
LIN {X 0,Y 375.589,Z 323.393,A -85,B 0,C 180,E1 14366.193,E2 14366.193} C_VEL
LIN {X 0,Y 384.388,Z 341.381,A -85,B 0,C 180,E1 14363.734,E2 14363.734} C_VEL
LIN {X 0,Y 385.03,Z 343.224,A -85,B 0,C 180,E1 14363.548,E2 14363.548} C_VEL
LIN {X 0,Y 373.644,Z 518.845,A -85,B 0,C 180,E1 14360.4,E2 14360.4} C_VEL
LIN {X 0,Y 371.532,Z 537.664,A -85,B 0,C 180,E1 14359.934,E2 14359.934} C_VEL
LIN {X 0,Y 367.915,Z 560.11,A -85,B 0,C 180,E1 14359.181,E2 14359.181} C_VEL
LIN {X 0,Y 363.726,Z 579.942,A -85,B 0,C 180,E1 14358.267,E2 14358.267} C_VEL
LIN {X 0,Y 359.382,Z 597.436,A -85,B 0,C 180,E1 14357.257,E2 14357.257} C_VEL
LIN {X 0,Y 354.879,Z 613.298,A -85,B 0,C 180,E1 14356.153,E2 14356.153} C_VEL
LIN {X 0,Y 349.996,Z 628.739,A -85,B 0,C 180,E1 14354.874,E2 14354.874} C_VEL
LIN {X 0,Y 344.789,Z 643.719,A -85,B 0,C 180,E1 14353.409,E2 14353.409} C_VEL
LIN {X 0,Y 338.859,Z 659.45,A -85,B 0,C 180,E1 14351.592,E2 14351.592} C_VEL
LIN {X 0,Y 331.285,Z 677.911,A -85,B 0,C 180,E1 14348.992,E2 14348.992} C_VEL
LIN {X 0,Y 325.335,Z 691.528,A -85,B 0,C 180,E1 14346.662,E2 14346.662} C_VEL
LIN {X 0,Y 320.253,Z 702.798,A -85,B 0,C 180,E1 14344.405,E2 14344.405} C_VEL
LIN {X 0,Y 315.435,Z 713.293,A -85,B 0,C 180,E1 14341.958,E2 14341.958} C_VEL
LIN {X 0,Y 310.883,Z 723.185,A -85,B 0,C 180,E1 14339.262,E2 14339.262} C_VEL
LIN {X 0,Y 306.736,Z 732.369,A -85,B 0,C 180,E1 14336.313,E2 14336.313} C_VEL
LIN {X 0,Y 302.768,Z 741.688,A -85,B 0,C 180,E1 14332.727,E2 14332.727} C_VEL
LIN {X 0,Y 299.401,Z 750.373,A -85,B 0,C 180,E1 14328.475,E2 14328.475} C_VEL
LIN {X 0,Y 297.602,Z 755.956,A -85,B 0,C 180,E1 14324.991,E2 14324.991} C_VEL
LIN {X 0,Y 296.575,Z 760.129,A -85,B 0,C 180,E1 14321.669,E2 14321.669} C_VEL
LIN {X 0,Y 296.073,Z 763.27,A -85,B 0,C 180,E1 14318.302,E2 14318.302} C_VEL
LIN {X 0,Y 295.943,Z 765.212,A -85,B 0,C 180,E1 14315.233,E2 14315.233} C_VEL
LIN {X 0,Y 295.965,Z 766.287,A -85,B 0,C 180,E1 14312.129,E2 14312.129} C_VEL
LIN {X 0,Y 295.976,Z 766.465,A -85,B 0,C 180,E1 14309.032,E2 14309.032} C_VEL
LIN {X 0,Y 295.946,Z 765.657,A -85,B 0,C 180,E1 14305.738,E2 14305.738} C_VEL
LIN {X 0,Y 296.039,Z 763.68,A -85,B 0,C 180,E1 14302.237,E2 14302.237} C_VEL
LIN {X 0,Y 296.448,Z 760.756,A -85,B 0,C 180,E1 14298.917,E2 14298.917} C_VEL
LIN {X 0,Y 297.397,Z 756.687,A -85,B 0,C 180,E1 14295.536,E2 14295.536} C_VEL
LIN {X 0,Y 298.94,Z 751.676,A -85,B 0,C 180,E1 14292.282,E2 14292.282} C_VEL
LIN {X 0,Y 301.236,Z 745.424,A -85,B 0,C 180,E1 14288.996,E2 14288.996} C_VEL
LIN {X 0,Y 304.313,Z 737.936,A -85,B 0,C 180,E1 14285.754,E2 14285.754} C_VEL
LIN {X 0,Y 308.987,Z 727.49,A -85,B 0,C 180,E1 14282.02,E2 14282.02} C_VEL
LIN {X 0,Y 314.476,Z 715.398,A -85,B 0,C 180,E1 14278.576,E2 14278.576} C_VEL
LIN {X 0,Y 319.534,Z 704.381,A -85,B 0,C 180,E1 14275.941,E2 14275.941} C_VEL
LIN {X 0,Y 324.817,Z 692.69,A -85,B 0,C 180,E1 14273.556,E2 14273.556} C_VEL
LIN {X 0,Y 330.419,Z 679.896,A -85,B 0,C 180,E1 14271.329,E2 14271.329} C_VEL
LIN {X 0,Y 336.256,Z 665.938,A -85,B 0,C 180,E1 14269.261,E2 14269.261} C_VEL
LIN {X 0,Y 343.525,Z 647.272,A -85,B 0,C 180,E1 14266.964,E2 14266.964} C_VEL
LIN {X 0,Y 349.466,Z 630.351,A -85,B 0,C 180,E1 14265.271,E2 14265.271} C_VEL
LIN {X 0,Y 354.556,Z 614.368,A -85,B 0,C 180,E1 14263.928,E2 14263.928} C_VEL
LIN {X 0,Y 359.126,Z 598.391,A -85,B 0,C 180,E1 14262.804,E2 14262.804} C_VEL
LIN {X 0,Y 363.222,Z 582.073,A -85,B 0,C 180,E1 14261.847,E2 14261.847} C_VEL
LIN {X 0,Y 366.819,Z 565.473,A -85,B 0,C 180,E1 14261.051,E2 14261.051} C_VEL
LIN {X 0,Y 370.114,Z 547.233,A -85,B 0,C 180,E1 14260.36,E2 14260.36} C_VEL
LIN {X 0,Y 373.238,Z 523.639,A -85,B 0,C 180,E1 14259.701,E2 14259.701} C_VEL
LIN {X 0,Y 375.827,Z 486.995,A -85,B 0,C 180,E1 14259.001,E2 14259.001} C_VEL
LIN {X 0,Y 384.978,Z 342.759,A -85,B 0,C 180,E1 14256.427,E2 14256.427} C_VEL
LIN {X 0,Y 376.877,Z 325.905,A -85,B 0,C 180,E1 14254.18,E2 14254.18} C_VEL
LIN {X 0,Y 368.36,Z 309.981,A -85,B 0,C 180,E1 14251.616,E2 14251.616} C_VEL
LIN {X 0,Y 361.825,Z 298.759,A -85,B 0,C 180,E1 14249.466,E2 14249.466} C_VEL
LIN {X 0,Y 358.198,Z 293.064,A -85,B 0,C 180,E1 14248.194,E2 14248.194} C_VEL
LIN {X 0,Y 351.371,Z 283.727,A -85,B 0,C 180,E1 14245.629,E2 14245.629} C_VEL
LIN {X 0,Y 347.864,Z 279.088,A -85,B 0,C 180,E1 14244.18,E2 14244.18} C_VEL
LIN {X 0,Y 344.207,Z 274.359,A -85,B 0,C 180,E1 14242.548,E2 14242.548} C_VEL
LIN {X 0,Y 340.01,Z 269.074,A -85,B 0,C 180,E1 14240.485,E2 14240.485} C_VEL
LIN {X 0,Y 336.539,Z 264.865,A -85,B 0,C 180,E1 14238.581,E2 14238.581} C_VEL
LIN {X 0,Y 335.516,Z 263.473,A -85,B 0,C 180,E1 14237.966,E2 14237.966} C_VEL
LIN {X 0,Y 332.129,Z 259.872,A -85,B 0,C 180,E1 14235.811,E2 14235.811} C_VEL
LIN {X 0,Y 330.917,Z 257.691,A -85,B 0,C 180,E1 14234.882,E2 14234.882} C_VEL
LIN {X 0,Y 327.48,Z 254.793,A -85,B 0,C 180,E1 14232.162,E2 14232.162} C_VEL
LIN {X 0,Y 325.721,Z 251.404,A -85,B 0,C 180,E1 14230.256,E2 14230.256} C_VEL
LIN {X 0,Y 320.949,Z 247.042,A -85,B 0,C 180,E1 14220.893,E2 14220.893} C_VEL
LIN {X 0,Y 321.053,Z 247.334,A -85,B 0,C 180,E1 14217.858,E2 14217.858} C_VEL
LIN {X 0,Y 325.838,Z 251.607,A -85,B 0,C 180,E1 14209.301,E2 14209.301} C_VEL
LIN {X 0,Y 328.003,Z 255.472,A -85,B 0,C 180,E1 14207.052,E2 14207.052} C_VEL
LIN {X 0,Y 331.141,Z 258.081,A -85,B 0,C 180,E1 14204.635,E2 14204.635} C_VEL
LIN {X 0,Y 333.94,Z 262.143,A -85,B 0,C 180,E1 14202.667,E2 14202.667} C_VEL
LIN {X 0,Y 336.216,Z 264.315,A -85,B 0,C 180,E1 14201.31,E2 14201.31} C_VEL
LIN {X 0,Y 339.559,Z 268.664,A -85,B 0,C 180,E1 14199.436,E2 14199.436} C_VEL
LIN {X 0,Y 341.122,Z 270.408,A -85,B 0,C 180,E1 14198.642,E2 14198.642} C_VEL
LIN {X 0,Y 345.908,Z 276.555,A -85,B 0,C 180,E1 14196.368,E2 14196.368} C_VEL
LIN {X 0,Y 349.984,Z 281.871,A -85,B 0,C 180,E1 14194.625,E2 14194.625} C_VEL
LIN {X 0,Y 356.799,Z 291.015,A -85,B 0,C 180,E1 14192.005,E2 14192.005} C_VEL
LIN {X 0,Y 365.506,Z 303.48,A -85,B 0,C 180,E1 14189.049,E2 14189.049} C_VEL
LIN {X 0,Y 376.991,Z 319.666,A -85,B 0,C 180,E1 14185.694,E2 14185.694} C_VEL
LIN {X 0,Y 388.937,Z 332.735,A -85,B 0,C 180,E1 14182.786,E2 14182.786} C_VEL
LIN {X 0,Y 397.974,Z 341.221,A -85,B 0,C 180,E1 14180.857,E2 14180.857} C_VEL
LIN {X 0,Y 407.481,Z 349.326,A -85,B 0,C 180,E1 14178.927,E2 14178.927} C_VEL
LIN {X 0,Y 415.447,Z 356.211,A -85,B 0,C 180,E1 14177.21,E2 14177.21} C_VEL
LIN {X 0,Y 424.676,Z 364.189,A -85,B 0,C 180,E1 14175.062,E2 14175.062} C_VEL
LIN {X 0,Y 432.719,Z 371.435,A -85,B 0,C 180,E1 14173.001,E2 14173.001} C_VEL
LIN {X 0,Y 441.191,Z 379.235,A -85,B 0,C 180,E1 14170.604,E2 14170.604} C_VEL
LIN {X 0,Y 449.692,Z 387.031,A -85,B 0,C 180,E1 14168.083,E2 14168.083} C_VEL
LIN {X 0,Y 458.519,Z 394.866,A -85,B 0,C 180,E1 14165.355,E2 14165.355} C_VEL
LIN {X 0,Y 463.817,Z 399.521,A -85,B 0,C 180,E1 14163.639,E2 14163.639} C_VEL
LIN {X 0,Y 471.795,Z 406.38,A -85,B 0,C 180,E1 14160.929,E2 14160.929} C_VEL
LIN {X 0,Y 477.841,Z 411.581,A -85,B 0,C 180,E1 14158.745,E2 14158.745} C_VEL
LIN {X 0,Y 481.352,Z 414.405,A -85,B 0,C 180,E1 14157.42,E2 14157.42} C_VEL
LIN {X 0,Y 486.846,Z 419.184,A -85,B 0,C 180,E1 14155.221,E2 14155.221} C_VEL
LIN {X 0,Y 491.204,Z 422.472,A -85,B 0,C 180,E1 14153.357,E2 14153.357} C_VEL
LIN {X 0,Y 495.925,Z 426.78,A -85,B 0,C 180,E1 14151.153,E2 14151.153} C_VEL
LIN {X 0,Y 500.677,Z 429.935,A -85,B 0,C 180,E1 14148.753,E2 14148.753} C_VEL
LIN {X 0,Y 504.823,Z 433.987,A -85,B 0,C 180,E1 14146.333,E2 14146.333} C_VEL
LIN {X 0,Y 508.349,Z 436.67,A -85,B 0,C 180,E1 14143.999,E2 14143.999} C_VEL
LIN {X 0,Y 511.676,Z 438.433,A -85,B 0,C 180,E1 14141.496,E2 14141.496} C_VEL
LIN {X 0,Y 512.701,Z 439.21,A -85,B 0,C 180,E1 14140.562,E2 14140.562} C_VEL
LIN {X 0,Y 514.836,Z 441.661,A -85,B 0,C 180,E1 14138.262,E2 14138.262} C_VEL
LIN {X 0,Y 516.452,Z 443.317,A -85,B 0,C 180,E1 14135.889,E2 14135.889} C_VEL
LIN {X 0,Y 517.7,Z 444.311,A -85,B 0,C 180,E1 14133.321,E2 14133.321} C_VEL
LIN {X 0,Y 518.2,Z 444.644,A -85,B 0,C 180,E1 14130.774,E2 14130.774} C_VEL
LIN {X 0,Y 518.086,Z 444.565,A -85,B 0,C 180,E1 14128.12,E2 14128.12} C_VEL
LIN {X 0,Y 517.23,Z 443.927,A -85,B 0,C 180,E1 14125.566,E2 14125.566} C_VEL
LIN {X 0,Y 515.677,Z 442.604,A -85,B 0,C 180,E1 14122.872,E2 14122.872} C_VEL
LIN {X 0,Y 513.504,Z 440.25,A -85,B 0,C 180,E1 14120.248,E2 14120.248} C_VEL
LIN {X 0,Y 511.939,Z 438.532,A -85,B 0,C 180,E1 14118.739,E2 14118.739} C_VEL
LIN {X 0,Y 508.527,Z 436.774,A -85,B 0,C 180,E1 14116.122,E2 14116.122} C_VEL
LIN {X 0,Y 505.024,Z 434.16,A -85,B 0,C 180,E1 14113.791,E2 14113.791} C_VEL
LIN {X 0,Y 501.161,Z 430.325,A -85,B 0,C 180,E1 14111.507,E2 14111.507} C_VEL
LIN {X 0,Y 496.228,Z 427.002,A -85,B 0,C 180,E1 14108.985,E2 14108.985} C_VEL
LIN {X 0,Y 491.445,Z 422.721,A -85,B 0,C 180,E1 14106.755,E2 14106.755} C_VEL
LIN {X 0,Y 488.717,Z 420.533,A -85,B 0,C 180,E1 14105.568,E2 14105.568} C_VEL
LIN {X 0,Y 483.044,Z 416.019,A -85,B 0,C 180,E1 14103.246,E2 14103.246} C_VEL
LIN {X 0,Y 478.908,Z 412.344,A -85,B 0,C 180,E1 14101.647,E2 14101.647} C_VEL
LIN {X 0,Y 472.763,Z 407.292,A -85,B 0,C 180,E1 14099.407,E2 14099.407} C_VEL
LIN {X 0,Y 468.287,Z 403.338,A -85,B 0,C 180,E1 14097.857,E2 14097.857} C_VEL
LIN {X 0,Y 461.597,Z 397.371,A -85,B 0,C 180,E1 14095.62,E2 14095.62} C_VEL
LIN {X 0,Y 453.873,Z 390.778,A -85,B 0,C 180,E1 14093.192,E2 14093.192} C_VEL
LIN {X 0,Y 444.782,Z 382.605,A -85,B 0,C 180,E1 14090.451,E2 14090.451} C_VEL
LIN {X 0,Y 435.494,Z 373.982,A -85,B 0,C 180,E1 14087.771,E2 14087.771} C_VEL
LIN {X 0,Y 427.337,Z 366.627,A -85,B 0,C 180,E1 14085.612,E2 14085.612} C_VEL
LIN {X 0,Y 418.773,Z 359.136,A -85,B 0,C 180,E1 14083.539,E2 14083.539} C_VEL
LIN {X 0,Y 409.158,Z 350.819,A -85,B 0,C 180,E1 14081.426,E2 14081.426} C_VEL
LIN {X 0,Y 399.43,Z 342.504,A -85,B 0,C 180,E1 14079.436,E2 14079.436} C_VEL
LIN {X 0,Y 389.21,Z 333.023,A -85,B 0,C 180,E1 14077.276,E2 14077.276} C_VEL
LIN {X 0,Y 376.991,Z 319.666,A -85,B 0,C 180,E1 14074.306,E2 14074.306} C_VEL
LIN {X 0,Y 365.506,Z 303.48,A -85,B 0,C 180,E1 14070.951,E2 14070.951} C_VEL
LIN {X 0,Y 356.401,Z 290.389,A -85,B 0,C 180,E1 14067.848,E2 14067.848} C_VEL
LIN {X 0,Y 348.248,Z 279.523,A -85,B 0,C 180,E1 14064.648,E2 14064.648} C_VEL
LIN {X 0,Y 344.137,Z 274.275,A -85,B 0,C 180,E1 14062.823,E2 14062.823} C_VEL
LIN {X 0,Y 340.105,Z 269.147,A -85,B 0,C 180,E1 14060.838,E2 14060.838} C_VEL
LIN {X 0,Y 336.616,Z 265.004,A -85,B 0,C 180,E1 14058.936,E2 14058.936} C_VEL
LIN {X 0,Y 335.741,Z 263.655,A -85,B 0,C 180,E1 14058.402,E2 14058.402} C_VEL
LIN {X 0,Y 332.312,Z 260.156,A -85,B 0,C 180,E1 14056.25,E2 14056.25} C_VEL
LIN {X 0,Y 330.744,Z 257.594,A -85,B 0,C 180,E1 14055.07,E2 14055.07} C_VEL
LIN {X 0,Y 327.437,Z 254.761,A -85,B 0,C 180,E1 14052.432,E2 14052.432} C_VEL
LIN {X 0,Y 325.598,Z 251.347,A -85,B 0,C 180,E1 14050.439,E2 14050.439} C_VEL
LIN {X 0,Y 320.95,Z 247.073,A -85,B 0,C 180,E1 14041.25,E2 14041.25} C_VEL
LIN {X 0,Y 321.072,Z 247.383,A -85,B 0,C 180,E1 14038.037,E2 14038.037} C_VEL
LIN {X 0,Y 325.866,Z 251.708,A -85,B 0,C 180,E1 14029.57,E2 14029.57} C_VEL
LIN {X 0,Y 328.146,Z 255.615,A -85,B 0,C 180,E1 14027.237,E2 14027.237} C_VEL
LIN {X 0,Y 331.135,Z 258.055,A -85,B 0,C 180,E1 14024.949,E2 14024.949} C_VEL
LIN {X 0,Y 333.864,Z 262.066,A -85,B 0,C 180,E1 14023.022,E2 14023.022} C_VEL
LIN {X 0,Y 336.207,Z 264.284,A -85,B 0,C 180,E1 14021.624,E2 14021.624} C_VEL
LIN {X 0,Y 339.533,Z 268.649,A -85,B 0,C 180,E1 14019.755,E2 14019.755} C_VEL
LIN {X 0,Y 341.104,Z 270.43,A -85,B 0,C 180,E1 14018.956,E2 14018.956} C_VEL
LIN {X 0,Y 345.749,Z 276.302,A -85,B 0,C 180,E1 14016.749,E2 14016.749} C_VEL
LIN {X 0,Y 347.346,Z 278.475,A -85,B 0,C 180,E1 14016.04,E2 14016.04} C_VEL
LIN {X 0,Y 349.658,Z 282.453,A -85,B 0,C 180,E1 14015.018,E2 14015.018} C_VEL
LIN {X 0,Y 352.636,Z 290.794,A -85,B 0,C 180,E1 14013.631,E2 14013.631} C_VEL
LIN {X 0,Y 356.041,Z 300.189,A -85,B 0,C 180,E1 14012.155,E2 14012.155} C_VEL
LIN {X 0,Y 356.73,Z 301.564,A -85,B 0,C 180,E1 14011.89,E2 14011.89} C_VEL
LIN {X 0,Y 364.178,Z 314.532,A -85,B 0,C 180,E1 14009.29,E2 14009.29} C_VEL
LIN {X 0,Y 372.18,Z 329.623,A -85,B 0,C 180,E1 14006.766,E2 14006.766} C_VEL
LIN {X 0,Y 380.108,Z 346.151,A -85,B 0,C 180,E1 14004.466,E2 14004.466} C_VEL
LIN {X 0,Y 368.584,Z 518.678,A -85,B 0,C 180,E1 14001.36,E2 14001.36} C_VEL
LIN {X 0,Y 366.403,Z 537.636,A -85,B 0,C 180,E1 14000.89,E2 14000.89} C_VEL
LIN {X 0,Y 362.56,Z 560.677,A -85,B 0,C 180,E1 14000.109,E2 14000.109} C_VEL
LIN {X 0,Y 358.423,Z 579.765,A -85,B 0,C 180,E1 13999.227,E2 13999.227} C_VEL
LIN {X 0,Y 353.965,Z 597.26,A -85,B 0,C 180,E1 13998.215,E2 13998.215} C_VEL
LIN {X 0,Y 349.34,Z 613.122,A -85,B 0,C 180,E1 13997.107,E2 13997.107} C_VEL
LIN {X 0,Y 344.315,Z 628.563,A -85,B 0,C 180,E1 13995.823,E2 13995.823} C_VEL
LIN {X 0,Y 338.953,Z 643.542,A -85,B 0,C 180,E1 13994.35,E2 13994.35} C_VEL
LIN {X 0,Y 332.831,Z 659.272,A -85,B 0,C 180,E1 13992.52,E2 13992.52} C_VEL
LIN {X 0,Y 325.057,Z 677.614,A -85,B 0,C 180,E1 13989.914,E2 13989.914} C_VEL
LIN {X 0,Y 319.122,Z 690.732,A -85,B 0,C 180,E1 13987.655,E2 13987.655} C_VEL
LIN {X 0,Y 313.551,Z 702.62,A -85,B 0,C 180,E1 13985.248,E2 13985.248} C_VEL
LIN {X 0,Y 308.53,Z 713.115,A -85,B 0,C 180,E1 13982.761,E2 13982.761} C_VEL
LIN {X 0,Y 303.775,Z 723.006,A -85,B 0,C 180,E1 13980.016,E2 13980.016} C_VEL
LIN {X 0,Y 299.426,Z 732.19,A -85,B 0,C 180,E1 13977.006,E2 13977.006} C_VEL
LIN {X 0,Y 295.245,Z 741.51,A -85,B 0,C 180,E1 13973.34,E2 13973.34} C_VEL
LIN {X 0,Y 291.689,Z 750.161,A -85,B 0,C 180,E1 13969.002,E2 13969.002} C_VEL
LIN {X 0,Y 289.752,Z 755.778,A -85,B 0,C 180,E1 13965.407,E2 13965.407} C_VEL
LIN {X 0,Y 288.643,Z 759.952,A -85,B 0,C 180,E1 13961.994,E2 13961.994} C_VEL
LIN {X 0,Y 288.098,Z 763.058,A -85,B 0,C 180,E1 13958.582,E2 13958.582} C_VEL
LIN {X 0,Y 287.947,Z 765.037,A -85,B 0,C 180,E1 13955.379,E2 13955.379} C_VEL
LIN {X 0,Y 287.965,Z 766.112,A -85,B 0,C 180,E1 13952.189,E2 13952.189} C_VEL
LIN {X 0,Y 287.978,Z 766.29,A -85,B 0,C 180,E1 13949.005,E2 13949.005} C_VEL
LIN {X 0,Y 287.945,Z 765.482,A -85,B 0,C 180,E1 13945.619,E2 13945.619} C_VEL
LIN {X 0,Y 288.049,Z 763.504,A -85,B 0,C 180,E1 13942.02,E2 13942.02} C_VEL
LIN {X 0,Y 288.506,Z 760.579,A -85,B 0,C 180,E1 13938.608,E2 13938.608} C_VEL
LIN {X 0,Y 289.508,Z 756.591,A -85,B 0,C 180,E1 13935.194,E2 13935.194} C_VEL
LIN {X 0,Y 291.183,Z 751.498,A -85,B 0,C 180,E1 13931.794,E2 13931.794} C_VEL
LIN {X 0,Y 293.623,Z 745.245,A -85,B 0,C 180,E1 13928.424,E2 13928.424} C_VEL
LIN {X 0,Y 296.876,Z 737.758,A -85,B 0,C 180,E1 13925.106,E2 13925.106} C_VEL
LIN {X 0,Y 301.787,Z 727.311,A -85,B 0,C 180,E1 13921.292,E2 13921.292} C_VEL
LIN {X 0,Y 307.532,Z 715.22,A -85,B 0,C 180,E1 13917.782,E2 13917.782} C_VEL
LIN {X 0,Y 312.802,Z 704.202,A -85,B 0,C 180,E1 13915.103,E2 13915.103} C_VEL
LIN {X 0,Y 318.292,Z 692.512,A -85,B 0,C 180,E1 13912.684,E2 13912.684} C_VEL
LIN {X 0,Y 324.098,Z 679.73,A -85,B 0,C 180,E1 13910.432,E2 13910.432} C_VEL
LIN {X 0,Y 330.143,Z 665.761,A -85,B 0,C 180,E1 13908.341,E2 13908.341} C_VEL
LIN {X 0,Y 337.681,Z 647.009,A -85,B 0,C 180,E1 13906.017,E2 13906.017} C_VEL
LIN {X 0,Y 343.768,Z 630.174,A -85,B 0,C 180,E1 13904.322,E2 13904.322} C_VEL
LIN {X 0,Y 348.839,Z 614.733,A -85,B 0,C 180,E1 13903.015,E2 13903.015} C_VEL
LIN {X 0,Y 353.379,Z 599.383,A -85,B 0,C 180,E1 13901.922,E2 13901.922} C_VEL
LIN {X 0,Y 357.518,Z 583.496,A -85,B 0,C 180,E1 13900.973,E2 13900.973} C_VEL
LIN {X 0,Y 361.313,Z 566.661,A -85,B 0,C 180,E1 13900.151,E2 13900.151} C_VEL
LIN {X 0,Y 364.537,Z 549.574,A -85,B 0,C 180,E1 13899.487,E2 13899.487} C_VEL
LIN {X 0,Y 367.202,Z 531.593,A -85,B 0,C 180,E1 13898.946,E2 13898.946} C_VEL
LIN {X 0,Y 369.415,Z 508.855,A -85,B 0,C 180,E1 13898.436,E2 13898.436} C_VEL
LIN {X 0,Y 380.018,Z 345.96,A -85,B 0,C 180,E1 13895.509,E2 13895.509} C_VEL
LIN {X 0,Y 371.664,Z 328.629,A -85,B 0,C 180,E1 13893.079,E2 13893.079} C_VEL
LIN {X 0,Y 363.963,Z 314.148,A -85,B 0,C 180,E1 13890.638,E2 13890.638} C_VEL
LIN {X 0,Y 356.387,Z 301.048,A -85,B 0,C 180,E1 13887.985,E2 13887.985} C_VEL
LIN {X 0,Y 349.015,Z 290.797,A -85,B 0,C 180,E1 13885.152,E2 13885.152} C_VEL
LIN {X 0,Y 345.454,Z 286.025,A -85,B 0,C 180,E1 13883.633,E2 13883.633} C_VEL
LIN {X 0,Y 342.053,Z 281.55,A -85,B 0,C 180,E1 13882.064,E2 13882.064} C_VEL
LIN {X 0,Y 338.11,Z 276.483,A -85,B 0,C 180,E1 13880.063,E2 13880.063} C_VEL
LIN {X 0,Y 334.598,Z 272.006,A -85,B 0,C 180,E1 13878.062,E2 13878.062} C_VEL
LIN {X 0,Y 333.036,Z 270.379,A -85,B 0,C 180,E1 13877.112,E2 13877.112} C_VEL
LIN {X 0,Y 330.006,Z 266.471,A -85,B 0,C 180,E1 13875.014,E2 13875.014} C_VEL
LIN {X 0,Y 329.246,Z 265.305,A -85,B 0,C 180,E1 13874.42,E2 13874.42} C_VEL
LIN {X 0,Y 325.96,Z 262.219,A -85,B 0,C 180,E1 13871.681,E2 13871.681} C_VEL
LIN {X 0,Y 324.418,Z 259.233,A -85,B 0,C 180,E1 13869.939,E2 13869.939} C_VEL
LIN {X 0,Y 319.973,Z 254.993,A -85,B 0,C 180,E1 13860.895,E2 13860.895} C_VEL
LIN {X 0,Y 320.077,Z 255.285,A -85,B 0,C 180,E1 13857.852,E2 13857.852} C_VEL
LIN {X 0,Y 324.612,Z 259.514,A -85,B 0,C 180,E1 13849.529,E2 13849.529} C_VEL
LIN {X 0,Y 326.74,Z 263.275,A -85,B 0,C 180,E1 13847.271,E2 13847.271} C_VEL
LIN {X 0,Y 329.697,Z 265.879,A -85,B 0,C 180,E1 13844.926,E2 13844.926} C_VEL
LIN {X 0,Y 332.582,Z 269.965,A -85,B 0,C 180,E1 13842.865,E2 13842.865} C_VEL
LIN {X 0,Y 334.543,Z 271.922,A -85,B 0,C 180,E1 13841.665,E2 13841.665} C_VEL
LIN {X 0,Y 338.047,Z 276.419,A -85,B 0,C 180,E1 13839.663,E2 13839.663} C_VEL
LIN {X 0,Y 339.655,Z 278.502,A -85,B 0,C 180,E1 13838.816,E2 13838.816} C_VEL
LIN {X 0,Y 343.831,Z 283.859,A -85,B 0,C 180,E1 13836.794,E2 13836.794} C_VEL
LIN {X 0,Y 347.981,Z 289.414,A -85,B 0,C 180,E1 13834.969,E2 13834.969} C_VEL
LIN {X 0,Y 354.593,Z 298.504,A -85,B 0,C 180,E1 13832.363,E2 13832.363} C_VEL
LIN {X 0,Y 362.741,Z 310.411,A -85,B 0,C 180,E1 13829.523,E2 13829.523} C_VEL
LIN {X 0,Y 374.427,Z 327.019,A -85,B 0,C 180,E1 13826.028,E2 13826.028} C_VEL
LIN {X 0,Y 389.834,Z 343.733,A -85,B 0,C 180,E1 13822.285,E2 13822.285} C_VEL
LIN {X 0,Y 404.703,Z 356.497,A -85,B 0,C 180,E1 13819.241,E2 13819.241} C_VEL
LIN {X 0,Y 413.421,Z 363.928,A -85,B 0,C 180,E1 13817.374,E2 13817.374} C_VEL
LIN {X 0,Y 421.325,Z 370.784,A -85,B 0,C 180,E1 13815.565,E2 13815.565} C_VEL
LIN {X 0,Y 430.518,Z 378.871,A -85,B 0,C 180,E1 13813.262,E2 13813.262} C_VEL
LIN {X 0,Y 438.611,Z 386.269,A -85,B 0,C 180,E1 13811.012,E2 13811.012} C_VEL
LIN {X 0,Y 447.86,Z 394.628,A -85,B 0,C 180,E1 13808.301,E2 13808.301} C_VEL
LIN {X 0,Y 456.944,Z 402.63,A -85,B 0,C 180,E1 13805.51,E2 13805.51} C_VEL
LIN {X 0,Y 465.001,Z 409.679,A -85,B 0,C 180,E1 13802.892,E2 13802.892} C_VEL
LIN {X 0,Y 470.203,Z 414.095,A -85,B 0,C 180,E1 13801.109,E2 13801.109} C_VEL
LIN {X 0,Y 476.503,Z 419.434,A -85,B 0,C 180,E1 13798.853,E2 13798.853} C_VEL
LIN {X 0,Y 479.99,Z 422.269,A -85,B 0,C 180,E1 13797.542,E2 13797.542} C_VEL
LIN {X 0,Y 485.575,Z 427.06,A -85,B 0,C 180,E1 13795.313,E2 13795.313} C_VEL
LIN {X 0,Y 489.899,Z 430.313,A -85,B 0,C 180,E1 13793.483,E2 13793.483} C_VEL
LIN {X 0,Y 494.647,Z 434.612,A -85,B 0,C 180,E1 13791.27,E2 13791.27} C_VEL
LIN {X 0,Y 499.592,Z 437.861,A -85,B 0,C 180,E1 13788.795,E2 13788.795} C_VEL
LIN {X 0,Y 503.765,Z 441.946,A -85,B 0,C 180,E1 13786.368,E2 13786.368} C_VEL
LIN {X 0,Y 507.312,Z 444.605,A -85,B 0,C 180,E1 13784.028,E2 13784.028} C_VEL
LIN {X 0,Y 510.668,Z 446.366,A -85,B 0,C 180,E1 13781.519,E2 13781.519} C_VEL
LIN {X 0,Y 511.81,Z 447.355,A -85,B 0,C 180,E1 13780.467,E2 13780.467} C_VEL
LIN {X 0,Y 514.011,Z 449.811,A -85,B 0,C 180,E1 13778.05,E2 13778.05} C_VEL
LIN {X 0,Y 515.551,Z 451.326,A -85,B 0,C 180,E1 13775.762,E2 13775.762} C_VEL
LIN {X 0,Y 516.799,Z 452.302,A -85,B 0,C 180,E1 13773.105,E2 13773.105} C_VEL
LIN {X 0,Y 517.251,Z 452.588,A -85,B 0,C 180,E1 13770.554,E2 13770.554} C_VEL
LIN {X 0,Y 517.025,Z 452.424,A -85,B 0,C 180,E1 13767.784,E2 13767.784} C_VEL
LIN {X 0,Y 516.161,Z 451.787,A -85,B 0,C 180,E1 13765.334,E2 13765.334} C_VEL
LIN {X 0,Y 514.595,Z 450.469,A -85,B 0,C 180,E1 13762.745,E2 13762.745} C_VEL
LIN {X 0,Y 512.454,Z 448.163,A -85,B 0,C 180,E1 13760.181,E2 13760.181} C_VEL
LIN {X 0,Y 510.888,Z 446.45,A -85,B 0,C 180,E1 13758.679,E2 13758.679} C_VEL
LIN {X 0,Y 507.49,Z 444.709,A -85,B 0,C 180,E1 13756.093,E2 13756.093} C_VEL
LIN {X 0,Y 503.967,Z 442.119,A -85,B 0,C 180,E1 13753.757,E2 13753.757} C_VEL
LIN {X 0,Y 499.992,Z 438.253,A -85,B 0,C 180,E1 13751.426,E2 13751.426} C_VEL
LIN {X 0,Y 494.943,Z 434.831,A -85,B 0,C 180,E1 13748.866,E2 13748.866} C_VEL
LIN {X 0,Y 490.148,Z 430.571,A -85,B 0,C 180,E1 13746.634,E2 13746.634} C_VEL
LIN {X 0,Y 487.073,Z 428.136,A -85,B 0,C 180,E1 13745.311,E2 13745.311} C_VEL
LIN {X 0,Y 481.388,Z 423.597,A -85,B 0,C 180,E1 13743.009,E2 13743.009} C_VEL
LIN {X 0,Y 477.402,Z 420.078,A -85,B 0,C 180,E1 13741.48,E2 13741.48} C_VEL
LIN {X 0,Y 471.22,Z 415.05,A -85,B 0,C 180,E1 13739.247,E2 13739.247} C_VEL
LIN {X 0,Y 466.497,Z 410.9,A -85,B 0,C 180,E1 13737.619,E2 13737.619} C_VEL
LIN {X 0,Y 459.578,Z 404.75,A -85,B 0,C 180,E1 13735.326,E2 13735.326} C_VEL
LIN {X 0,Y 451.972,Z 398.308,A -85,B 0,C 180,E1 13732.948,E2 13732.948} C_VEL
LIN {X 0,Y 442.592,Z 389.902,A -85,B 0,C 180,E1 13730.135,E2 13730.135} C_VEL
LIN {X 0,Y 433.559,Z 381.635,A -85,B 0,C 180,E1 13727.561,E2 13727.561} C_VEL
LIN {X 0,Y 425.835,Z 374.792,A -85,B 0,C 180,E1 13725.546,E2 13725.546} C_VEL
LIN {X 0,Y 419.887,Z 369.626,A -85,B 0,C 180,E1 13724.103,E2 13724.103} C_VEL
LIN {X 0,Y 410.314,Z 361.404,A -85,B 0,C 180,E1 13721.937,E2 13721.937} C_VEL
LIN {X 0,Y 399.604,Z 352.403,A -85,B 0,C 180,E1 13719.741,E2 13719.741} C_VEL
